C01783=1043.976,340.554,-119.354,172.680,41.723,158.046
C01784=1043.968,340.306,-119.318,172.674,41.720,158.045
C01785=1043.961,340.060,-119.281,172.670,41.717,158.044
C01786=1043.954,339.812,-119.244,172.665,41.714,158.043
C01787=1043.946,339.565,-119.208,172.660,41.710,158.041
C01788=1043.939,339.317,-119.172,172.656,41.707,158.040
C01789=1043.932,339.070,-119.136,172.650,41.703,158.039
C01790=1043.925,338.823,-119.099,172.646,41.700,158.038
C01791=1043.917,338.576,-119.063,172.641,41.697,158.037
C01792=1043.911,338.328,-119.027,172.636,41.693,158.036
C01793=1043.903,338.081,-118.990,172.631,41.690,158.035
C01794=1043.896,337.834,-118.955,172.627,41.686,158.034
C01795=1043.888,337.587,-118.918,172.622,41.683,158.033
C01796=1043.882,337.340,-118.882,172.618,41.680,158.032
C01797=1043.874,337.092,-118.846,172.612,41.677,158.031
C01798=1043.866,336.845,-118.810,172.608,41.673,158.030
C01799=1043.860,336.598,-118.773,172.603,41.670,158.029
C01800=1043.853,336.350,-118.738,172.599,41.667,158.028
C01801=1043.846,336.103,-118.702,172.593,41.663,158.026
C01802=1043.838,335.855,-118.665,172.589,41.660,158.026
C01803=1043.832,335.608,-118.629,172.584,41.657,158.025
C01804=1043.824,335.361,-118.593,172.580,41.653,158.023
C01805=1043.817,335.114,-118.558,172.575,41.650,158.022
C01806=1043.810,334.866,-118.521,172.571,41.647,158.021
C01807=1043.802,334.619,-118.486,172.565,41.644,158.020
C01808=1043.795,334.371,-118.450,172.561,41.640,158.019
C01809=1043.785,334.043,-118.402,172.555,41.636,158.018
C01810=1043.776,333.714,-118.355,172.549,41.632,158.017
C01811=1043.766,333.386,-118.307,172.543,41.628,158.015
C01812=1043.756,333.058,-118.260,172.537,41.623,158.014
C01813=1043.749,332.811,-118.225,172.532,41.620,158.013
C01814=1043.742,332.564,-118.189,172.528,41.617,158.012
C01815=1043.736,332.315,-118.153,172.522,41.614,158.011
C01816=1043.728,332.069,-118.117,172.518,41.611,158.010
C01817=1043.721,331.821,-118.081,172.514,41.608,158.009
C01818=1043.714,331.573,-118.046,172.509,41.605,158.008
C01819=1043.707,331.326,-118.010,172.505,41.602,158.007
C01820=1043.700,331.078,-117.975,172.500,41.599,158.006
C01821=1043.693,330.832,-117.939,172.495,41.595,158.005
C01822=1043.686,330.584,-117.904,172.491,41.592,158.004
C01823=1043.679,330.336,-117.868,172.486,41.589,158.003
C01824=1043.672,330.090,-117.833,172.482,41.586,158.002
C01825=1043.665,329.842,-117.797,172.478,41.583,158.001
C01826=1043.657,329.594,-117.762,172.473,41.580,158.000
C01827=1043.650,329.347,-117.726,172.469,41.577,157.999
C01828=1043.643,329.100,-117.692,172.465,41.573,157.998
C01829=1043.635,328.852,-117.656,172.459,41.570,157.997
C01830=1043.629,328.605,-117.621,172.456,41.568,157.996
C01831=1043.621,328.358,-117.586,172.450,41.565,157.995
C01832=1043.614,328.110,-117.551,172.446,41.562,157.994
C01833=1043.607,327.862,-117.516,172.442,41.558,157.993
C01834=1043.600,327.615,-117.481,172.437,41.556,157.993
C01835=1043.592,327.367,-117.446,172.433,41.553,157.992
C01836=1043.585,327.120,-117.411,172.429,41.550,157.991
C01837=1043.578,326.873,-117.376,172.424,41.547,157.990
C01838=1043.571,326.625,-117.341,172.420,41.544,157.989
C01839=1043.563,326.378,-117.306,172.416,41.541,157.988
C01840=1043.556,326.130,-117.271,172.411,41.538,157.987
C01841=1043.549,325.883,-117.236,172.407,41.535,157.986
C01842=1043.541,325.635,-117.201,172.403,41.532,157.985
C01843=1043.534,325.388,-117.166,172.398,41.529,157.984
C01844=1043.527,325.141,-117.131,172.393,41.526,157.983
C01845=1043.520,324.893,-117.096,172.389,41.524,157.982
C01846=1043.513,324.646,-117.061,172.384,41.521,157.981
C01847=1043.506,324.398,-117.027,172.380,41.517,157.980
C01848=1043.498,324.151,-116.992,172.376,41.515,157.980
C01849=1043.492,323.903,-116.957,172.372,41.512,157.979
C01850=1043.485,323.656,-116.922,172.367,41.509,157.978
C01851=1043.477,323.409,-116.887,172.363,41.506,157.977
C01852=1043.471,323.161,-116.853,172.359,41.503,157.976
C01853=1043.463,322.914,-116.818,172.355,41.500,157.975
C01854=1043.456,322.666,-116.783,172.350,41.497,157.974
C01855=1043.449,322.418,-116.749,172.346,41.494,157.973
C01856=1043.442,322.171,-116.714,172.342,41.492,157.972
C01857=1043.434,321.924,-116.679,172.338,41.488,157.971
C01858=1043.428,321.676,-116.645,172.333,41.486,157.970
C01859=1043.420,321.429,-116.610,172.329,41.483,157.969
C01860=1043.414,321.181,-116.575,172.325,41.480,157.969
C01861=1043.407,320.933,-116.541,172.321,41.477,157.968
C01862=1043.400,320.686,-116.506,172.317,41.474,157.967
C01863=1043.393,320.438,-116.472,172.312,41.471,157.966
C01864=1043.386,320.191,-116.437,172.308,41.469,157.965
C01865=1043.376,319.858,-116.391,172.302,41.465,157.964
C01866=1043.367,319.524,-116.344,172.297,41.461,157.963
C01867=1043.358,319.191,-116.298,172.291,41.457,157.962
C01868=1043.348,318.858,-116.251,172.285,41.453,157.960
C01869=1043.342,318.611,-116.218,172.281,41.451,157.959
C01870=1043.335,318.363,-116.183,172.277,41.447,157.958
C01871=1043.328,318.116,-116.149,172.273,41.445,157.958
C01872=1043.321,317.868,-116.114,172.268,41.442,157.957
C01873=1043.314,317.621,-116.080,172.264,41.439,157.956
C01874=1043.307,317.373,-116.045,172.260,41.437,157.955
C01875=1043.300,317.126,-116.011,172.256,41.433,157.954
C01876=1043.293,316.878,-115.976,172.252,41.431,157.953
C01877=1043.286,316.630,-115.943,172.248,41.428,157.952
C01878=1043.280,316.383,-115.909,172.244,41.425,157.952
C01879=1043.273,316.136,-115.874,172.240,41.423,157.951
C01880=1043.266,315.888,-115.840,172.236,41.419,157.950
C01881=1043.259,315.640,-115.806,172.231,41.417,157.949
C01882=1043.252,315.392,-115.771,172.227,41.414,157.948
C01883=1043.245,315.145,-115.737,172.223,41.411,157.947
C01884=1043.239,314.898,-115.703,172.219,41.409,157.946
C01885=1043.232,314.650,-115.669,172.215,41.406,157.946
C01886=1043.225,314.402,-115.634,172.211,41.403,157.945
C01887=1043.218,314.154,-115.601,172.207,41.400,157.944
C01888=1043.212,313.908,-115.566,172.204,41.398,157.943
C01889=1043.205,313.660,-115.532,172.200,41.395,157.942
C01890=1043.198,313.412,-115.498,172.196,41.392,157.941
C01891=1043.191,313.164,-115.464,172.192,41.389,157.940
C01892=1043.185,312.917,-115.430,172.188,41.387,157.940
C01893=1043.178,312.669,-115.396,172.184,41.383,157.939
C01894=1043.171,312.422,-115.362,172.180,41.381,157.938
C01895=1043.164,312.175,-115.329,172.176,41.378,157.937
C01896=1043.157,311.927,-115.295,172.171,41.376,157.936
C01897=1043.150,311.679,-115.261,172.167,41.373,157.935
C01898=1043.143,311.432,-115.227,172.163,41.371,157.935
C01899=1043.136,311.183,-115.194,172.159,41.368,157.934
C01900=1043.129,310.936,-115.161,172.155,41.365,157.933
C01901=1043.122,310.689,-115.127,172.151,41.363,157.932
C01902=1043.115,310.441,-115.093,172.147,41.360,157.931
C01903=1043.108,310.193,-115.060,172.143,41.358,157.931
C01904=1043.101,309.946,-115.027,172.140,41.355,157.930
C01905=1043.093,309.698,-114.993,172.136,41.352,157.929
C01906=1043.086,309.451,-114.959,172.132,41.350,157.928
C01907=1043.080,309.203,-114.927,172.128,41.348,157.927
C01908=1043.073,308.955,-114.893,172.124,41.345,157.927
C01909=1043.066,308.708,-114.859,172.120,41.343,157.926
C01910=1043.059,308.459,-114.826,172.116,41.340,157.925
C01911=1043.052,308.212,-114.792,172.112,41.337,157.924
C01912=1043.044,307.965,-114.759,172.108,41.335,157.923
C01913=1043.038,307.718,-114.726,172.105,41.332,157.923
C01914=1043.031,307.470,-114.693,172.101,41.330,157.922
C01915=1043.024,307.222,-114.659,172.097,41.327,157.921
C01916=1043.017,306.975,-114.626,172.093,41.325,157.920
C01917=1043.010,306.726,-114.593,172.089,41.322,157.920
C01918=1043.003,306.479,-114.559,172.085,41.320,157.919
C01919=1042.996,306.232,-114.526,172.081,41.317,157.918
C01920=1042.989,305.984,-114.493,172.077,41.314,157.917
C01921=1042.980,305.655,-114.449,172.072,41.311,157.916
C01922=1042.971,305.326,-114.405,172.067,41.308,157.915
C01923=1042.962,304.998,-114.361,172.062,41.305,157.914
C01924=1042.953,304.669,-114.317,172.057,41.302,157.913
C01925=1042.946,304.422,-114.284,172.053,41.299,157.912
C01926=1042.939,304.174,-114.251,172.049,41.296,157.911
C01927=1042.933,303.926,-114.218,172.045,41.294,157.911
C01928=1042.925,303.679,-114.185,172.041,41.291,157.910
C01929=1042.919,303.431,-114.152,172.038,41.289,157.909
C01930=1042.912,303.183,-114.119,172.034,41.286,157.908
C01931=1042.905,302.936,-114.085,172.030,41.284,157.908
C01932=1042.898,302.688,-114.052,172.026,41.281,157.907
C01933=1042.892,302.440,-114.019,172.023,41.279,157.906
C01934=1042.884,302.193,-113.986,172.019,41.277,157.905
C01935=1042.878,301.945,-113.954,172.015,41.274,157.905
C01936=1042.871,301.697,-113.921,172.011,41.271,157.904
C01937=1042.864,301.449,-113.888,172.008,41.269,157.903
C01938=1042.858,301.202,-113.854,172.004,41.267,157.902
C01939=1042.850,300.954,-113.822,172.000,41.264,157.902
C01940=1042.844,300.707,-113.789,171.996,41.261,157.901
C01941=1042.838,300.459,-113.756,171.992,41.259,157.900
C01942=1042.831,300.211,-113.723,171.989,41.257,157.899
C01943=1042.824,299.963,-113.690,171.985,41.254,157.899
C01944=1042.816,299.716,-113.657,171.982,41.252,157.898
C01945=1042.810,299.468,-113.624,171.978,41.249,157.897
C01946=1042.804,299.221,-113.592,171.974,41.247,157.896
C01947=1042.797,298.972,-113.559,171.970,41.244,157.895
C01948=1042.791,298.725,-113.526,171.967,41.242,157.895
C01949=1042.784,298.477,-113.494,171.963,41.239,157.894
C01950=1042.777,298.229,-113.461,171.960,41.237,157.893
C01951=1042.770,297.981,-113.428,171.956,41.235,157.893
C01952=1042.764,297.734,-113.395,171.952,41.232,157.892
C01953=1042.758,297.486,-113.362,171.948,41.229,157.891
C01954=1042.750,297.238,-113.330,171.945,41.227,157.890
C01955=1042.744,296.991,-113.297,171.941,41.225,157.890
C01956=1042.738,296.743,-113.264,171.938,41.223,157.889
C01957=1042.731,296.496,-113.232,171.934,41.220,157.888
C01958=1042.724,296.248,-113.199,171.930,41.217,157.887
C01959=1042.717,296.000,-113.166,171.927,41.215,157.887
C01960=1042.711,295.752,-113.134,171.923,41.213,157.886
C01961=1042.705,295.504,-113.102,171.919,41.210,157.885
C01962=1042.698,295.256,-113.069,171.916,41.208,157.884
C01963=1042.691,295.009,-113.037,171.913,41.206,157.884
C01964=1042.684,294.761,-113.004,171.909,41.203,157.883
C01965=1042.678,294.513,-112.973,171.905,41.201,157.882
C01966=1042.671,294.265,-112.940,171.901,41.198,157.882
C01967=1042.664,294.018,-112.907,171.898,41.196,157.881
C01968=1042.658,293.770,-112.875,171.895,41.194,157.880
C01969=1042.651,293.522,-112.843,171.891,41.192,157.879
C01970=1042.644,293.274,-112.810,171.887,41.189,157.879
C01971=1042.637,293.026,-112.779,171.884,41.187,157.878
C01972=1042.630,292.779,-112.747,171.881,41.185,157.877
C01973=1042.624,292.531,-112.714,171.877,41.182,157.877
C01974=1042.616,292.283,-112.682,171.873,41.180,157.876
C01975=1042.609,292.035,-112.650,171.869,41.177,157.875
C01976=1042.603,291.787,-112.618,171.866,41.175,157.875
C01977=1042.594,291.475,-112.577,171.862,41.173,157.874
C01978=1042.586,291.163,-112.538,171.858,41.170,157.873
C01979=1042.578,290.851,-112.497,171.853,41.167,157.872
C01980=1042.569,290.539,-112.456,171.849,41.164,157.871
C01981=1042.562,290.290,-112.424,171.845,41.162,157.870
C01982=1042.556,290.042,-112.392,171.841,41.159,157.870
C01983=1042.549,289.795,-112.360,171.837,41.157,157.869
C01984=1042.542,289.547,-112.329,171.835,41.155,157.868
C01985=1042.535,289.300,-112.297,171.831,41.153,157.868
C01986=1042.529,289.052,-112.265,171.827,41.150,157.867
C01987=1042.522,288.804,-112.233,171.824,41.148,157.866
C01988=1042.515,288.556,-112.201,171.821,41.146,157.866
C01989=1042.508,288.308,-112.169,171.817,41.143,157.865
C01990=1042.501,288.060,-112.138,171.814,41.141,157.864
C01991=1042.495,287.812,-112.105,171.810,41.139,157.864
C01992=1042.488,287.564,-112.074,171.807,41.137,157.863
C01993=1042.482,287.316,-112.042,171.803,41.135,157.862
C01994=1042.475,287.069,-112.011,171.800,41.132,157.861
C01995=1042.468,286.821,-111.979,171.796,41.130,157.861
C01996=1042.461,286.573,-111.947,171.793,41.128,157.860
C01997=1042.454,286.325,-111.916,171.790,41.126,157.860
C01998=1042.448,286.077,-111.884,171.786,41.123,157.859
C01999=1042.442,285.829,-111.852,171.782,41.121,157.858
C02000=1042.434,285.581,-111.821,171.780,41.119,157.857
C02001=1042.427,285.333,-111.788,171.776,41.117,157.857
C02002=1042.421,285.086,-111.757,171.772,41.115,157.856
C02003=1042.414,284.838,-111.725,171.770,41.113,157.856
C02004=1042.407,284.590,-111.694,171.766,41.110,157.855
C02005=1042.400,284.342,-111.663,171.762,41.108,157.854
C02006=1042.394,284.094,-111.631,171.759,41.106,157.854
C02007=1042.387,283.846,-111.600,171.755,41.104,157.853
C02008=1042.380,283.598,-111.568,171.752,41.102,157.852
C02009=1042.373,283.350,-111.537,171.749,41.100,157.852
C02010=1042.367,283.102,-111.505,171.745,41.098,157.851
C02011=1042.360,282.854,-111.474,171.743,41.096,157.850
C02012=1042.353,282.607,-111.443,171.739,41.093,157.850
C02013=1042.347,282.359,-111.411,171.735,41.091,157.849
C02014=1042.340,282.111,-111.380,171.732,41.089,157.848
C02015=1042.333,281.863,-111.348,171.729,41.087,157.848
C02016=1042.326,281.615,-111.317,171.726,41.084,157.847
C02017=1042.320,281.366,-111.286,171.722,41.082,157.846
C02018=1042.314,281.119,-111.255,171.719,41.080,157.846
C02019=1042.307,280.871,-111.224,171.716,41.078,157.845
C02020=1042.300,280.623,-111.192,171.712,41.076,157.844
C02021=1042.294,280.376,-111.161,171.709,41.073,157.844
C02022=1042.287,280.128,-111.129,171.706,41.071,157.843
C02023=1042.280,279.880,-111.098,171.702,41.069,157.842
C02024=1042.274,279.631,-111.067,171.699,41.067,157.842
C02025=1042.267,279.383,-111.036,171.695,41.065,157.841
C02026=1042.260,279.135,-111.004,171.693,41.063,157.841
C02027=1042.254,278.888,-110.973,171.689,41.061,157.840
C02028=1042.248,278.640,-110.943,171.686,41.059,157.839
C02029=1042.240,278.392,-110.912,171.683,41.057,157.839
C02030=1042.234,278.144,-110.880,171.679,41.054,157.838
C02031=1042.227,277.896,-110.850,171.676,41.052,157.837
C02032=1042.220,277.648,-110.818,171.673,41.050,157.837
C02033=1042.212,277.348,-110.781,171.669,41.048,157.836
C02034=1042.204,277.047,-110.743,171.665,41.045,157.835
C02035=1042.196,276.747,-110.706,171.661,41.043,157.834
C02036=1042.187,276.446,-110.669,171.657,41.040,157.834
C02037=1042.181,276.198,-110.637,171.654,41.038,157.833
C02038=1042.175,275.950,-110.607,171.651,41.036,157.832
C02039=1042.168,275.702,-110.575,171.647,41.034,157.832
C02040=1042.161,275.454,-110.545,171.644,41.032,157.831
C02041=1042.154,275.206,-110.514,171.641,41.030,157.831
C02042=1042.148,274.958,-110.483,171.638,41.027,157.830
C02043=1042.142,274.710,-110.452,171.634,41.025,157.829
C02044=1042.135,274.462,-110.422,171.632,41.023,157.829
C02045=1042.128,274.214,-110.391,171.628,41.021,157.828
C02046=1042.121,273.966,-110.360,171.625,41.020,157.828
C02047=1042.114,273.718,-110.329,171.622,41.017,157.827
C02048=1042.108,273.470,-110.299,171.619,41.015,157.826
C02049=1042.101,273.223,-110.268,171.615,41.013,157.826
C02050=1042.094,272.974,-110.237,171.613,41.011,157.825
C02051=1042.088,272.726,-110.206,171.609,41.009,157.824
C02052=1042.081,272.479,-110.176,171.606,41.007,157.824
C02053=1042.075,272.230,-110.145,171.603,41.005,157.823
C02054=1042.068,271.982,-110.114,171.600,41.003,157.822
C02055=1042.061,271.734,-110.084,171.596,41.001,157.822
C02056=1042.055,271.486,-110.053,171.594,40.999,157.821
C02057=1042.049,271.238,-110.023,171.591,40.997,157.821
C02058=1042.041,270.990,-109.992,171.587,40.995,157.820
C02059=1042.035,270.742,-109.961,171.585,40.992,157.819
C02060=1042.028,270.494,-109.931,171.581,40.990,157.819
C02061=1042.022,270.246,-109.901,171.578,40.989,157.818
C02062=1042.014,269.998,-109.870,171.575,40.987,157.818
C02063=1042.009,269.750,-109.840,171.572,40.984,157.817
C02064=1042.001,269.502,-109.809,171.568,40.982,157.816
C02065=1041.995,269.254,-109.778,171.566,40.980,157.816
C02066=1041.988,269.005,-109.748,171.562,40.979,157.815
C02067=1041.982,268.758,-109.718,171.559,40.977,157.815
C02068=1041.975,268.509,-109.688,171.557,40.974,157.814
C02069=1041.968,268.261,-109.658,171.553,40.972,157.813
C02070=1041.962,268.013,-109.627,171.550,40.970,157.813
C02071=1041.955,267.765,-109.597,171.547,40.969,157.812
C02072=1041.949,267.517,-109.567,171.544,40.966,157.812
C02073=1041.942,267.269,-109.537,171.540,40.964,157.811
C02074=1041.935,267.021,-109.506,171.538,40.962,157.811
C02075=1041.929,266.773,-109.476,171.535,40.961,157.810
C02076=1041.921,266.525,-109.446,171.531,40.959,157.809
C02077=1041.915,266.276,-109.415,171.529,40.956,157.809
C02078=1041.908,266.029,-109.386,171.525,40.954,157.808
C02079=1041.901,265.781,-109.356,171.523,40.953,157.808
C02080=1041.895,265.532,-109.325,171.520,40.950,157.807
C02081=1041.888,265.285,-109.295,171.516,40.948,157.806
C02082=1041.881,265.036,-109.265,171.514,40.946,157.806
C02083=1041.875,264.788,-109.235,171.510,40.945,157.805
C02084=1041.868,264.540,-109.205,171.507,40.943,157.805
C02085=1041.861,264.292,-109.174,171.505,40.940,157.804
C02086=1041.855,264.044,-109.144,171.501,40.939,157.804
C02087=1041.848,263.795,-109.115,171.498,40.937,157.803
C02088=1041.842,263.548,-109.085,171.496,40.934,157.802
C02089=1041.833,263.252,-109.048,171.492,40.932,157.802
C02090=1041.826,262.956,-109.013,171.488,40.930,157.801
C02091=1041.818,262.660,-108.977,171.484,40.928,157.800
C02092=1041.810,262.364,-108.941,171.481,40.925,157.800
C02093=1041.803,262.116,-108.912,171.478,40.923,157.799
C02094=1041.797,261.868,-108.882,171.475,40.921,157.798
C02095=1041.790,261.620,-108.852,171.472,40.920,157.798
C02096=1041.783,261.372,-108.823,171.469,40.917,157.797
C02097=1041.776,261.123,-108.793,171.466,40.916,157.797
C02098=1041.769,260.875,-108.763,171.463,40.914,157.796
C02099=1041.763,260.627,-108.733,171.461,40.912,157.796
C02100=1041.756,260.379,-108.703,171.457,40.910,157.795
C02101=1041.750,260.131,-108.674,171.454,40.908,157.794
C02102=1041.742,259.883,-108.644,171.452,40.906,157.794
C02103=1041.736,259.634,-108.615,171.448,40.904,157.793
C02104=1041.729,259.386,-108.585,171.445,40.903,157.793
C02105=1041.723,259.138,-108.556,171.443,40.900,157.792
C02106=1041.715,258.890,-108.526,171.439,40.899,157.792
C02107=1041.708,258.641,-108.497,171.437,40.897,157.791
C02108=1041.701,258.394,-108.467,171.434,40.895,157.791
C02109=1041.695,258.145,-108.438,171.430,40.893,157.790
C02110=1041.688,257.898,-108.408,171.428,40.891,157.790
C02111=1041.681,257.649,-108.379,171.425,40.889,157.789
C02112=1041.675,257.401,-108.349,171.422,40.888,157.788
C02113=1041.668,257.153,-108.320,171.419,40.886,157.788
C02114=1041.661,256.905,-108.290,171.416,40.884,157.787
C02115=1041.655,256.657,-108.261,171.413,40.882,157.787
C02116=1041.648,256.408,-108.231,171.410,40.880,157.786
C02117=1041.642,256.160,-108.202,171.408,40.878,157.786
C02118=1041.635,255.912,-108.172,171.405,40.876,157.785
C02119=1041.627,255.664,-108.143,171.401,40.874,157.785
C02120=1041.621,255.415,-108.114,171.399,40.872,157.784
C02121=1041.614,255.167,-108.085,171.396,40.871,157.784
C02122=1041.608,254.920,-108.055,171.393,40.868,157.783
C02123=1041.601,254.671,-108.025,171.390,40.867,157.782
C02124=1041.595,254.423,-107.996,171.387,40.865,157.782
C02125=1041.587,254.175,-107.966,171.385,40.863,157.781
C02126=1041.581,253.927,-107.937,171.382,40.861,157.781
C02127=1041.575,253.678,-107.908,171.379,40.859,157.780
C02128=1041.568,253.430,-107.879,171.376,40.857,157.780
C02129=1041.562,253.182,-107.849,171.373,40.855,157.779
C02130=1041.554,252.934,-107.820,171.371,40.853,157.779
C02131=1041.548,252.685,-107.791,171.367,40.852,157.778
C02132=1041.541,252.437,-107.762,171.365,40.850,157.777
C02133=1041.535,252.188,-107.733,171.362,40.847,157.777
C02134=1041.528,251.941,-107.703,171.359,40.846,157.776
C02135=1041.522,251.693,-107.674,171.356,40.844,157.776
C02136=1041.515,251.444,-107.644,171.353,40.842,157.775
C02137=1041.509,251.196,-107.615,171.350,40.840,157.775
C02138=1041.502,250.948,-107.587,171.348,40.838,157.774
C02139=1041.495,250.701,-107.557,171.345,40.836,157.774
C02140=1041.488,250.452,-107.528,171.342,40.835,157.773
C02141=1041.482,250.204,-107.499,171.339,40.832,157.772
C02142=1041.476,249.955,-107.470,171.337,40.831,157.772
C02143=1041.469,249.707,-107.440,171.334,40.828,157.771
C02144=1041.463,249.458,-107.411,171.331,40.827,157.771
C02145=1041.455,249.161,-107.376,171.328,40.824,157.770
C02146=1041.447,248.864,-107.342,171.324,40.822,157.770
C02147=1041.439,248.567,-107.307,171.321,40.820,157.769
C02148=1041.431,248.269,-107.272,171.318,40.818,157.768
C02149=1041.425,248.021,-107.243,171.315,40.816,157.768
C02150=1041.418,247.772,-107.214,171.312,40.814,157.767
C02151=1041.412,247.524,-107.185,171.310,40.812,157.767
C02152=1041.406,247.276,-107.156,171.307,40.810,157.766
C02153=1041.399,247.028,-107.127,171.304,40.808,157.766
C02154=1041.392,246.780,-107.098,171.301,40.806,157.765
C02155=1041.386,246.531,-107.069,171.298,40.804,157.764
C02156=1041.380,246.283,-107.040,171.296,40.802,157.764
C02157=1041.373,246.035,-107.011,171.293,40.800,157.763
C02158=1041.367,245.787,-106.982,171.290,40.798,157.763
C02159=1041.360,245.539,-106.953,171.288,40.796,157.762
C02160=1041.353,245.290,-106.924,171.285,40.794,157.762
C02161=1041.347,245.042,-106.896,171.283,40.793,157.761
C02162=1041.341,244.793,-106.866,171.279,40.791,157.761
C02163=1041.334,244.546,-106.838,171.277,40.789,157.760
C02164=1041.328,244.298,-106.809,171.274,40.787,157.759
C02165=1041.320,244.049,-106.780,171.271,40.785,157.759
C02166=1041.314,243.800,-106.752,171.269,40.783,157.759
C02167=1041.308,243.552,-106.723,171.266,40.781,157.758
C02168=1041.301,243.304,-106.694,171.264,40.780,157.757
C02169=1041.295,243.056,-106.665,171.261,40.777,157.757
C02170=1041.288,242.808,-106.638,171.259,40.776,157.756
C02171=1041.281,242.559,-106.608,171.255,40.774,157.756
C02172=1041.275,242.311,-106.579,171.252,40.772,157.755
C02173=1041.268,242.062,-106.551,171.250,40.770,157.755
C02174=1041.262,241.814,-106.522,171.247,40.768,157.754
C02175=1041.255,241.566,-106.494,171.245,40.767,157.754
C02176=1041.249,241.318,-106.466,171.242,40.764,157.753
C02177=1041.242,241.070,-106.437,171.240,40.763,157.753
C02178=1041.235,240.821,-106.408,171.237,40.761,157.752
C02179=1041.229,240.573,-106.380,171.234,40.759,157.752
C02180=1041.222,240.324,-106.351,171.232,40.757,157.751
C02181=1041.216,240.076,-106.323,171.229,40.755,157.751
C02182=1041.209,239.828,-106.295,171.226,40.754,157.750
C02183=1041.203,239.579,-106.266,171.223,40.752,157.750
C02184=1041.196,239.332,-106.238,171.221,40.750,157.749
C02185=1041.188,239.082,-106.210,171.218,40.748,157.749
C02186=1041.182,238.834,-106.181,171.215,40.747,157.748
C02187=1041.176,238.586,-106.153,171.213,40.744,157.747
C02188=1041.169,238.338,-106.125,171.210,40.743,157.747
C02189=1041.163,238.089,-106.096,171.208,40.741,157.747
C02190=1041.156,237.841,-106.068,171.205,40.739,157.746
C02191=1041.149,237.593,-106.040,171.203,40.737,157.745
C02192=1041.143,237.345,-106.011,171.200,40.736,157.745
C02193=1041.136,237.096,-105.983,171.197,40.733,157.744
C02194=1041.129,236.848,-105.956,171.195,40.732,157.744
C02195=1041.122,236.600,-105.927,171.192,40.730,157.743
C02196=1041.116,236.351,-105.899,171.190,40.728,157.743
C02197=1041.109,236.103,-105.870,171.187,40.726,157.742
C02198=1041.102,235.854,-105.842,171.185,40.725,157.742
C02199=1041.095,235.606,-105.815,171.181,40.723,157.741
C02200=1041.089,235.358,-105.786,171.179,40.721,157.741
C02201=1041.081,235.054,-105.752,171.176,40.719,157.740
C02202=1041.073,234.752,-105.718,171.173,40.716,157.740
C02203=1041.065,234.449,-105.684,171.170,40.714,157.739
C02204=1041.057,234.146,-105.649,171.167,40.712,157.738
C02205=1041.051,233.897,-105.621,171.164,40.710,157.738
C02206=1041.044,233.649,-105.593,171.162,40.708,157.737
C02207=1041.037,233.401,-105.565,171.159,40.707,157.737
C02208=1041.031,233.152,-105.537,171.157,40.704,157.736
C02209=1041.025,232.904,-105.509,171.154,40.703,157.736
C02210=1041.018,232.655,-105.481,171.152,40.701,157.735
C02211=1041.011,232.407,-105.452,171.149,40.699,157.735
C02212=1041.004,232.159,-105.425,171.147,40.697,157.734
C02213=1040.998,231.910,-105.396,171.144,40.696,157.734
C02214=1040.992,231.662,-105.369,171.141,40.693,157.733
C02215=1040.985,231.413,-105.341,171.139,40.692,157.733
C02216=1040.978,231.165,-105.313,171.136,40.690,157.732
C02217=1040.972,230.916,-105.286,171.134,40.688,157.732
C02218=1040.965,230.669,-105.257,171.131,40.686,157.731
C02219=1040.958,230.420,-105.229,171.129,40.685,157.731
C02220=1040.951,230.172,-105.202,171.126,40.682,157.730
C02221=1040.945,229.923,-105.174,171.124,40.681,157.730
C02222=1040.939,229.675,-105.146,171.121,40.679,157.729
C02223=1040.932,229.426,-105.118,171.118,40.677,157.729
C02224=1040.925,229.178,-105.090,171.116,40.675,157.728
C02225=1040.919,228.929,-105.062,171.113,40.674,157.728
C02226=1040.913,228.681,-105.035,171.111,40.672,157.727
C02227=1040.906,228.433,-105.007,171.108,40.670,157.727
C02228=1040.899,228.185,-104.980,171.106,40.668,157.726
C02229=1040.893,227.936,-104.952,171.103,40.667,157.726
C02230=1040.886,227.688,-104.924,171.102,40.665,157.725
C02231=1040.879,227.439,-104.896,171.099,40.663,157.725
C02232=1040.872,227.191,-104.869,171.097,40.661,157.724
C02233=1040.865,226.943,-104.841,171.094,40.659,157.724
C02234=1040.858,226.694,-104.814,171.092,40.658,157.723
C02235=1040.852,226.445,-104.787,171.089,40.655,157.723
C02236=1040.845,226.197,-104.759,171.086,40.654,157.722
C02237=1040.839,225.948,-104.731,171.084,40.652,157.722
C02238=1040.833,225.701,-104.704,171.081,40.651,157.721
C02239=1040.826,225.452,-104.676,171.079,40.648,157.721
C02240=1040.818,225.204,-104.649,171.076,40.647,157.720
C02241=1040.812,224.956,-104.621,171.074,40.645,157.720
C02242=1040.805,224.706,-104.594,171.071,40.643,157.719
C02243=1040.799,224.458,-104.567,171.070,40.641,157.719
C02244=1040.792,224.210,-104.539,171.067,40.639,157.718
C02245=1040.785,223.961,-104.511,171.065,40.638,157.718
C02246=1040.779,223.713,-104.484,171.062,40.636,157.717
C02247=1040.772,223.465,-104.457,171.060,40.634,157.717
C02248=1040.766,223.216,-104.430,171.057,40.632,157.716
C02249=1040.759,222.968,-104.402,171.055,40.631,157.716
C02250=1040.752,222.719,-104.374,171.052,40.629,157.715
C02251=1040.746,222.471,-104.347,171.049,40.627,157.715
C02252=1040.740,222.223,-104.320,171.048,40.625,157.714
C02253=1040.732,221.974,-104.293,171.045,40.623,157.714
C02254=1040.726,221.725,-104.266,171.043,40.621,157.713
C02255=1040.719,221.477,-104.238,171.040,40.620,157.713
C02256=1040.713,221.229,-104.211,171.038,40.618,157.712
C02257=1040.704,220.918,-104.176,171.035,40.616,157.712
C02258=1040.697,220.608,-104.142,171.032,40.613,157.711
C02259=1040.688,220.297,-104.108,171.029,40.611,157.711
C02260=1040.680,219.987,-104.074,171.026,40.608,157.710
C02261=1040.674,219.738,-104.047,171.024,40.607,157.709
C02262=1040.666,219.490,-104.020,171.021,40.605,157.709
C02263=1040.660,219.240,-103.993,171.019,40.603,157.708
C02264=1040.653,218.992,-103.965,171.017,40.602,157.708
C02265=1040.647,218.745,-103.939,171.015,40.600,157.708
C02266=1040.640,218.496,-103.912,171.012,40.598,157.707
C02267=1040.633,218.247,-103.884,171.009,40.596,157.706
C02268=1040.626,217.998,-103.857,171.007,40.595,157.706
C02269=1040.620,217.751,-103.831,171.004,40.593,157.706
C02270=1040.613,217.502,-103.804,171.003,40.591,157.705
C02271=1040.607,217.253,-103.777,171.000,40.589,157.705
C02272=1040.599,217.005,-103.749,170.998,40.587,157.704
C02273=1040.594,216.756,-103.723,170.995,40.586,157.704
C02274=1040.586,216.508,-103.696,170.993,40.584,157.703
C02275=1040.580,216.259,-103.669,170.991,40.582,157.703
C02276=1040.572,216.011,-103.642,170.989,40.580,157.702
C02277=1040.567,215.763,-103.615,170.986,40.578,157.702
C02278=1040.560,215.514,-103.588,170.984,40.577,157.701
C02279=1040.553,215.265,-103.561,170.981,40.575,157.701
C02280=1040.547,215.017,-103.534,170.980,40.573,157.700
C02281=1040.540,214.769,-103.507,170.977,40.571,157.700
C02282=1040.533,214.520,-103.480,170.975,40.569,157.699
C02283=1040.527,214.272,-103.454,170.972,40.568,157.699
C02284=1040.520,214.023,-103.426,170.969,40.566,157.698
C02285=1040.513,213.775,-103.400,170.968,40.564,157.698
C02286=1040.507,213.526,-103.373,170.965,40.562,157.697
C02287=1040.500,213.278,-103.345,170.963,40.561,157.697
C02288=1040.493,213.029,-103.319,170.960,40.558,157.696
C02289=1040.488,212.781,-103.292,170.959,40.557,157.696
C02290=1040.480,212.533,-103.265,170.956,40.555,157.695
C02291=1040.474,212.284,-103.238,170.954,40.553,157.695
C02292=1040.467,212.035,-103.212,170.951,40.551,157.694
C02293=1040.461,211.786,-103.185,170.950,40.549,157.694
C02294=1040.454,211.539,-103.158,170.947,40.548,157.693
C02295=1040.448,211.290,-103.131,170.945,40.546,157.693
C02296=1040.441,211.041,-103.105,170.942,40.544,157.692
C02297=1040.434,210.793,-103.079,170.941,40.542,157.692
C02298=1040.428,210.544,-103.052,170.938,40.540,157.691
C02299=1040.420,210.296,-103.025,170.936,40.539,157.691
C02300=1040.415,210.048,-102.998,170.933,40.537,157.691
C02301=1040.407,209.799,-102.972,170.932,40.535,157.690
C02302=1040.401,209.551,-102.946,170.929,40.533,157.689
C02303=1040.395,209.302,-102.919,170.927,40.531,157.689
C02304=1040.387,209.053,-102.892,170.925,40.530,157.689
C02305=1040.381,208.805,-102.866,170.923,40.528,157.688
C02306=1040.375,208.556,-102.839,170.920,40.526,157.688
C02307=1040.368,208.308,-102.813,170.918,40.524,157.687
C02308=1040.361,208.060,-102.786,170.916,40.522,157.687
C02309=1040.353,207.811,-102.759,170.914,40.521,157.686
C02310=1040.348,207.563,-102.733,170.911,40.519,157.686
C02311=1040.341,207.314,-102.706,170.909,40.517,157.685
C02312=1040.334,207.066,-102.680,170.907,40.515,157.685
C02313=1040.326,206.760,-102.648,170.904,40.513,157.684
C02314=1040.318,206.455,-102.616,170.902,40.510,157.684
C02315=1040.310,206.150,-102.583,170.899,40.509,157.683
C02316=1040.301,205.845,-102.551,170.896,40.507,157.682
C02317=1040.275,204.794,-102.445,170.609,40.403,157.648
C02318=1040.269,204.545,-102.419,170.606,40.402,157.648
C02319=1040.263,204.296,-102.394,170.602,40.401,157.647
C02320=1040.256,204.048,-102.369,170.599,40.400,157.647
C02321=1040.250,203.799,-102.343,170.597,40.399,157.647
C02322=1040.245,203.551,-102.318,170.593,40.397,157.646
C02323=1040.239,203.302,-102.294,170.590,40.397,157.646
C02324=1040.233,203.053,-102.268,170.587,40.395,157.646
C02325=1040.226,202.805,-102.244,170.584,40.395,157.645
C02326=1040.219,202.556,-102.218,170.581,40.394,157.645
C02327=1040.213,202.307,-102.193,170.578,40.393,157.645
C02328=1040.208,202.059,-102.169,170.575,40.392,157.644
C02329=1040.202,201.810,-102.143,170.572,40.391,157.644
C02330=1040.195,201.561,-102.118,170.569,40.390,157.644
C02331=1040.189,201.313,-102.093,170.566,40.388,157.643
C02332=1040.183,201.063,-102.068,170.563,40.387,157.643
C02333=1040.176,200.815,-102.043,170.560,40.386,157.643
C02334=1040.170,200.566,-102.018,170.557,40.385,157.642
C02335=1040.165,200.318,-101.994,170.554,40.385,157.642
C02336=1040.158,200.069,-101.969,170.551,40.384,157.642
C02337=1040.152,199.820,-101.944,170.548,40.383,157.641
C02338=1040.145,199.572,-101.920,170.545,40.382,157.641
C02339=1040.139,199.323,-101.895,170.542,40.381,157.641
C02340=1040.133,199.074,-101.870,170.539,40.380,157.640
C02341=1040.127,198.826,-101.846,170.536,40.379,157.640
C02342=1040.121,198.577,-101.821,170.533,40.378,157.640
C02343=1040.114,198.329,-101.796,170.530,40.377,157.639
C02344=1040.108,198.079,-101.771,170.527,40.377,157.639
C02345=1040.101,197.831,-101.747,170.525,40.376,157.639
C02346=1040.096,197.582,-101.722,170.521,40.375,157.638
C02347=1040.090,197.333,-101.698,170.518,40.374,157.638
C02348=1040.083,197.085,-101.673,170.516,40.373,157.638
C02349=1040.077,196.835,-101.648,170.512,40.372,157.637
C02350=1040.070,196.587,-101.624,170.510,40.371,157.637
C02351=1040.065,196.338,-101.599,170.507,40.370,157.637
C02352=1040.058,196.090,-101.575,170.503,40.370,157.637
C02353=1040.052,195.841,-101.550,170.501,40.368,157.636
C02354=1040.046,195.593,-101.526,170.498,40.368,157.636
C02355=1040.040,195.344,-101.501,170.494,40.367,157.636
C02356=1040.033,195.095,-101.477,170.492,40.366,157.635
C02357=1040.027,194.846,-101.452,170.489,40.365,157.635
C02358=1040.021,194.598,-101.427,170.487,40.364,157.635
C02359=1040.015,194.349,-101.403,170.483,40.363,157.634
C02360=1040.009,194.100,-101.378,170.480,40.362,157.634
C02361=1040.003,193.852,-101.354,170.478,40.361,157.634
C02362=1039.997,193.602,-101.330,170.474,40.360,157.633
C02363=1039.990,193.354,-101.305,170.472,40.360,157.633
C02364=1039.984,193.105,-101.281,170.469,40.359,157.633
C02365=1039.978,192.856,-101.257,170.466,40.358,157.633
C02366=1039.972,192.607,-101.232,170.463,40.357,157.632
C02367=1039.966,192.360,-101.208,170.460,40.356,157.632
C02368=1039.960,192.110,-101.183,170.458,40.356,157.632
C02369=1039.953,191.861,-101.159,170.454,40.355,157.631
C02370=1039.948,191.613,-101.135,170.452,40.354,157.631
C02371=1039.941,191.364,-101.110,170.449,40.353,157.631
C02372=1039.935,191.116,-101.086,170.445,40.352,157.630
C02373=1039.929,190.867,-101.062,170.443,40.351,157.630
C02374=1039.923,190.617,-101.037,170.440,40.350,157.630
C02375=1039.918,190.369,-101.013,170.438,40.349,157.630
C02376=1039.911,190.121,-100.988,170.434,40.348,157.629
C02377=1039.905,189.872,-100.964,170.432,40.348,157.629
C02378=1039.898,189.587,-100.936,170.429,40.347,157.629
C02379=1039.891,189.303,-100.908,170.425,40.346,157.628
C02380=1039.884,189.018,-100.881,170.422,40.345,157.628
C02381=1039.877,188.734,-100.853,170.419,40.344,157.628
C02382=1039.871,188.485,-100.829,170.416,40.343,157.627
C02383=1039.865,188.237,-100.805,170.413,40.342,157.627
C02384=1039.859,187.988,-100.780,170.411,40.341,157.627
C02385=1039.853,187.739,-100.757,170.408,40.341,157.627
C02386=1039.847,187.490,-100.732,170.405,40.340,157.626
C02387=1039.841,187.242,-100.708,170.402,40.339,157.626
C02388=1039.835,186.992,-100.684,170.400,40.338,157.626
C02389=1039.829,186.744,-100.660,170.396,40.337,157.625
C02390=1039.824,186.495,-100.636,170.394,40.336,157.625
C02391=1039.817,186.247,-100.612,170.391,40.335,157.625
C02392=1039.812,185.997,-100.587,170.388,40.334,157.624
C02393=1039.806,185.749,-100.564,170.385,40.334,157.624
C02394=1039.799,185.500,-100.540,170.383,40.333,157.624
C02395=1039.794,185.252,-100.515,170.380,40.332,157.624
C02396=1039.787,185.003,-100.491,170.377,40.332,157.623
C02397=1039.782,184.754,-100.467,170.374,40.331,157.623
C02398=1039.775,184.505,-100.443,170.372,40.330,157.623
C02399=1039.770,184.256,-100.419,170.369,40.329,157.622
C02400=1039.764,184.008,-100.395,170.366,40.328,157.622
C02401=1039.758,183.759,-100.371,170.363,40.327,157.622
C02402=1039.752,183.511,-100.347,170.361,40.326,157.622
C02403=1039.745,183.261,-100.324,170.358,40.326,157.621
C02404=1039.739,183.013,-100.300,170.355,40.325,157.621
C02405=1039.733,182.764,-100.276,170.352,40.325,157.621
C02406=1039.727,182.515,-100.252,170.350,40.324,157.621
C02407=1039.720,182.266,-100.229,170.347,40.323,157.620
C02408=1039.714,182.018,-100.205,170.344,40.323,157.620
C02409=1039.708,181.769,-100.181,170.341,40.322,157.620
C02410=1039.702,181.520,-100.158,170.339,40.321,157.620
C02411=1039.695,181.271,-100.135,170.336,40.321,157.619
C02412=1039.689,181.023,-100.111,170.333,40.320,157.619
C02413=1039.682,180.773,-100.088,170.330,40.320,157.619
C02414=1039.676,180.525,-100.064,170.328,40.319,157.619
C02415=1039.670,180.276,-100.040,170.325,40.318,157.618
C02416=1039.664,180.027,-100.017,170.323,40.318,157.618
C02417=1039.657,179.778,-99.993,170.319,40.317,157.618
C02418=1039.651,179.529,-99.970,170.317,40.316,157.618
C02419=1039.645,179.280,-99.946,170.314,40.316,157.618
C02420=1039.639,179.032,-99.923,170.312,40.315,157.617
C02421=1039.632,178.783,-99.900,170.308,40.315,157.617
C02422=1039.626,178.534,-99.876,170.306,40.314,157.617
C02423=1039.620,178.285,-99.853,170.303,40.313,157.617
C02424=1039.613,178.036,-99.829,170.301,40.313,157.616
C02425=1039.608,177.788,-99.806,170.297,40.313,157.616
C02426=1039.601,177.539,-99.782,170.295,40.312,157.616
C02427=1039.595,177.290,-99.759,170.292,40.311,157.616
C02428=1039.589,177.041,-99.736,170.290,40.310,157.615
C02429=1039.583,176.792,-99.712,170.288,40.310,157.615
C02430=1039.576,176.544,-99.689,170.284,40.309,157.615
C02431=1039.570,176.294,-99.666,170.282,40.308,157.615
C02432=1039.564,176.046,-99.642,170.279,40.308,157.614
C02433=1039.558,175.797,-99.619,170.277,40.308,157.614
C02434=1039.551,175.548,-99.595,170.273,40.307,157.614
C02435=1039.546,175.299,-99.572,170.271,40.306,157.614
C02436=1039.540,175.050,-99.549,170.268,40.306,157.614
C02437=1039.533,174.801,-99.525,170.266,40.305,157.613
C02438=1039.527,174.553,-99.503,170.264,40.304,157.613
C02439=1039.521,174.304,-99.479,170.260,40.304,157.613
C02440=1039.514,174.055,-99.456,170.258,40.303,157.613
C02441=1039.509,173.806,-99.433,170.255,40.303,157.612
C02442=1039.502,173.521,-99.406,170.253,40.302,157.612
C02443=1039.495,173.237,-99.380,170.249,40.301,157.612
C02444=1039.488,172.952,-99.353,170.246,40.301,157.612
C02445=1039.481,172.667,-99.327,170.243,40.300,157.611
C02446=1039.474,172.418,-99.303,170.241,40.300,157.611
C02447=1039.468,172.169,-99.280,170.238,40.299,157.611
C02448=1039.463,171.921,-99.257,170.235,40.298,157.611
C02449=1039.456,171.672,-99.235,170.233,40.298,157.610
C02450=1039.450,171.423,-99.211,170.230,40.297,157.610
C02451=1039.444,171.174,-99.188,170.227,40.296,157.610
C02452=1039.438,170.925,-99.165,170.225,40.296,157.610
C02453=1039.432,170.676,-99.142,170.222,40.295,157.609
C02454=1039.426,170.427,-99.118,170.220,40.295,157.609
C02455=1039.420,170.178,-99.095,170.217,40.294,157.609
C02456=1039.414,169.930,-99.073,170.214,40.294,157.609
C02457=1039.408,169.681,-99.050,170.212,40.293,157.608
C02458=1039.401,169.432,-99.026,170.209,40.293,157.608
C02459=1039.395,169.183,-99.003,170.207,40.292,157.608
C02460=1039.390,168.934,-98.980,170.205,40.291,157.608
C02461=1039.383,168.686,-98.957,170.201,40.291,157.608
C02462=1039.378,168.437,-98.934,170.199,40.290,157.607
C02463=1039.371,168.188,-98.911,170.197,40.289,157.607
C02464=1039.365,167.939,-98.887,170.194,40.289,157.607
C02465=1039.359,167.690,-98.864,170.191,40.288,157.607
C02466=1039.354,167.441,-98.842,170.189,40.288,157.607
C02467=1039.347,167.192,-98.819,170.186,40.287,157.606
C02468=1039.342,166.944,-98.796,170.184,40.287,157.606
C02469=1039.336,166.695,-98.773,170.182,40.286,157.606
C02470=1039.329,166.445,-98.750,170.178,40.285,157.605
C02471=1039.324,166.196,-98.727,170.176,40.285,157.605
C02472=1039.317,165.948,-98.704,170.174,40.284,157.605
C02473=1039.311,165.699,-98.681,170.171,40.283,157.605
C02474=1039.305,165.450,-98.658,170.169,40.283,157.605
C02475=1039.300,165.201,-98.635,170.166,40.283,157.604
C02476=1039.294,164.953,-98.612,170.163,40.282,157.604
C02477=1039.288,164.704,-98.590,170.161,40.281,157.604
C02478=1039.282,164.455,-98.567,170.159,40.281,157.604
C02479=1039.275,164.205,-98.544,170.155,40.280,157.604
C02480=1039.270,163.957,-98.521,170.153,40.279,157.603
C02481=1039.264,163.708,-98.498,170.151,40.279,157.603
C02482=1039.258,163.459,-98.475,170.149,40.279,157.603
C02483=1039.252,163.210,-98.452,170.146,40.278,157.603
C02484=1039.246,162.961,-98.429,170.143,40.277,157.602
C02485=1039.240,162.712,-98.406,170.141,40.277,157.602
C02486=1039.234,162.464,-98.384,170.138,40.276,157.602
C02487=1039.228,162.215,-98.361,170.136,40.275,157.602
C02488=1039.222,161.966,-98.338,170.134,40.275,157.601
C02489=1039.217,161.717,-98.315,170.131,40.274,157.601
C02490=1039.211,161.468,-98.293,170.128,40.274,157.601
C02491=1039.205,161.219,-98.271,170.126,40.273,157.601
C02492=1039.199,160.970,-98.248,170.124,40.273,157.601
C02493=1039.193,160.721,-98.225,170.122,40.272,157.600
C02494=1039.188,160.472,-98.202,170.118,40.272,157.600
C02495=1039.181,160.224,-98.180,170.116,40.271,157.600
C02496=1039.175,159.975,-98.157,170.114,40.270,157.600
C02497=1039.169,159.726,-98.135,170.111,40.270,157.600
C02498=1039.164,159.477,-98.112,170.109,40.270,157.599
C02499=1039.157,159.228,-98.090,170.106,40.269,157.599
C02500=1039.151,158.979,-98.067,170.104,40.269,157.599
C02501=1039.145,158.729,-98.045,170.101,40.268,157.599
C02502=1039.138,158.481,-98.022,170.099,40.268,157.599
C02503=1039.132,158.232,-97.999,170.097,40.268,157.598
C02504=1039.126,157.983,-97.978,170.093,40.267,157.598
C02505=1039.120,157.734,-97.955,170.091,40.267,157.598
C02506=1039.113,157.449,-97.930,170.088,40.266,157.598
C02507=1039.106,157.164,-97.904,170.086,40.265,157.598
C02508=1039.100,156.878,-97.879,170.083,40.265,157.597
C02509=1039.092,156.593,-97.853,170.080,40.265,157.597
C02510=1039.086,156.345,-97.830,170.077,40.264,157.597
C02511=1039.080,156.096,-97.809,170.075,40.264,157.597
C02512=1039.074,155.847,-97.786,170.073,40.263,157.597
C02513=1039.068,155.597,-97.764,170.070,40.263,157.596
C02514=1039.062,155.349,-97.741,170.068,40.263,157.596
C02515=1039.056,155.100,-97.719,170.065,40.262,157.596
C02516=1039.049,154.851,-97.697,170.063,40.262,157.596
C02517=1039.044,154.602,-97.674,170.060,40.261,157.596
C02518=1039.038,154.353,-97.653,170.058,40.260,157.595
C02519=1039.031,154.104,-97.630,170.056,40.260,157.595
C02520=1039.025,153.855,-97.609,170.053,40.259,157.595
C02521=1039.019,153.606,-97.586,170.050,40.259,157.595
C02522=1039.013,153.357,-97.564,170.048,40.259,157.595
C02523=1039.007,153.108,-97.542,170.046,40.259,157.595
C02524=1039.000,152.859,-97.520,170.044,40.258,157.594
C02525=1038.994,152.610,-97.498,170.041,40.258,157.594
C02526=1038.989,152.361,-97.476,170.039,40.258,157.594
C02527=1038.982,152.112,-97.453,170.036,40.257,157.594
C02528=1038.976,151.864,-97.432,170.034,40.257,157.594
C02529=1038.970,151.615,-97.410,170.031,40.257,157.593
C02530=1038.964,151.366,-97.388,170.029,40.256,157.593
C02531=1038.958,151.116,-97.366,170.027,40.256,157.593
C02532=1038.952,150.868,-97.343,170.025,40.255,157.593
C02533=1038.946,150.619,-97.322,170.021,40.255,157.593
C02534=1038.939,150.370,-97.299,170.019,40.254,157.593
C02535=1038.933,150.121,-97.278,170.017,40.254,157.592
C02536=1038.928,149.871,-97.256,170.015,40.254,157.592
C02537=1038.921,149.623,-97.233,170.012,40.253,157.592
C02538=1038.915,149.374,-97.212,170.010,40.253,157.592
C02539=1038.910,149.125,-97.190,170.007,40.252,157.592
C02540=1038.903,148.876,-97.168,170.005,40.252,157.591
C02541=1038.897,148.627,-97.146,170.003,40.252,157.591
C02542=1038.891,148.378,-97.125,170.000,40.251,157.591
C02543=1038.885,148.129,-97.102,169.998,40.251,157.591
C02544=1038.879,147.880,-97.080,169.996,40.250,157.591
C02545=1038.873,147.631,-97.058,169.993,40.250,157.591
C02546=1038.867,147.382,-97.037,169.990,40.250,157.590
C02547=1038.861,147.134,-97.015,169.988,40.250,157.590
C02548=1038.854,146.884,-96.993,169.986,40.249,157.590
C02549=1038.848,146.635,-96.972,169.984,40.249,157.590
C02550=1038.842,146.386,-96.950,169.982,40.248,157.590
C02551=1038.836,146.137,-96.928,169.978,40.248,157.590
C02552=1038.830,145.888,-96.906,169.976,40.248,157.589
C02553=1038.823,145.639,-96.884,169.974,40.247,157.589
C02554=1038.818,145.391,-96.863,169.972,40.247,157.589
C02555=1038.812,145.141,-96.841,169.969,40.247,157.589
C02556=1038.805,144.892,-96.820,169.967,40.247,157.589
C02557=1038.799,144.643,-96.799,169.965,40.246,157.589
C02558=1038.792,144.394,-96.777,169.962,40.246,157.588
C02559=1038.786,144.145,-96.755,169.960,40.245,157.588
C02560=1038.780,143.897,-96.733,169.957,40.245,157.588
C02561=1038.774,143.648,-96.712,169.955,40.245,157.588
C02562=1038.768,143.399,-96.690,169.953,40.245,157.588
C02563=1038.762,143.149,-96.669,169.951,40.244,157.588
C02564=1038.756,142.900,-96.647,169.949,40.244,157.587
C02565=1038.750,142.652,-96.626,169.945,40.244,157.587
C02566=1038.744,142.402,-96.604,169.943,40.243,157.587
C02567=1038.738,142.153,-96.582,169.941,40.243,157.587
C02568=1038.732,141.904,-96.561,169.939,40.243,157.587
C02569=1038.726,141.655,-96.539,169.937,40.242,157.587
C02570=1038.718,141.370,-96.515,169.934,40.242,157.586
C02571=1038.712,141.085,-96.490,169.932,40.242,157.586
C02572=1038.705,140.799,-96.465,169.928,40.241,157.586
C02573=1038.697,140.514,-96.441,169.926,40.241,157.586
C02574=1038.691,140.265,-96.419,169.924,40.240,157.586
C02575=1038.685,140.015,-96.398,169.921,40.240,157.586
C02576=1038.679,139.766,-96.376,169.919,40.240,157.585
C02577=1038.673,139.518,-96.355,169.917,40.239,157.585
C02578=1038.667,139.268,-96.333,169.915,40.239,157.585
C02579=1038.661,139.019,-96.312,169.912,40.239,157.585
C02580=1038.654,138.770,-96.291,169.910,40.239,157.585
C02581=1038.649,138.521,-96.270,169.907,40.238,157.585
C02582=1038.643,138.272,-96.248,169.905,40.238,157.585
C02583=1038.637,138.023,-96.226,169.903,40.238,157.584
C02584=1038.630,137.774,-96.205,169.901,40.238,157.584
C02585=1038.624,137.525,-96.184,169.898,40.237,157.584
C02586=1038.618,137.276,-96.163,169.896,40.237,157.584
C02587=1038.612,137.026,-96.142,169.893,40.237,157.584
C02588=1038.606,136.778,-96.121,169.891,40.237,157.584
C02589=1038.600,136.529,-96.099,169.889,40.236,157.583
C02590=1038.593,136.280,-96.078,169.887,40.236,157.583
C02591=1038.587,136.031,-96.057,169.885,40.236,157.583
C02592=1038.581,135.782,-96.036,169.883,40.235,157.583
C02593=1038.575,135.533,-96.014,169.879,40.235,157.583
C02594=1038.568,135.284,-95.993,169.877,40.235,157.583
C02595=1038.563,135.035,-95.972,169.875,40.235,157.583
C02596=1038.557,134.786,-95.950,169.873,40.234,157.582
C02597=1038.550,134.536,-95.930,169.871,40.234,157.582
C02598=1038.544,134.288,-95.909,169.869,40.234,157.582
C02599=1038.538,134.039,-95.887,169.866,40.234,157.582
C02600=1038.531,133.790,-95.866,169.864,40.233,157.582
C02601=1038.526,133.541,-95.846,169.861,40.233,157.582
C02602=1038.520,133.291,-95.824,169.859,40.233,157.581
C02603=1038.513,133.043,-95.803,169.857,40.233,157.581
C02604=1038.508,132.793,-95.782,169.855,40.232,157.581
C02605=1038.501,132.545,-95.761,169.853,40.232,157.581
C02606=1038.495,132.296,-95.740,169.850,40.231,157.581
C02607=1038.489,132.046,-95.719,169.848,40.232,157.581
C02608=1038.483,131.797,-95.698,169.845,40.231,157.581
C02609=1038.477,131.549,-95.677,169.843,40.231,157.580
C02610=1038.471,131.299,-95.656,169.841,40.230,157.580
C02611=1038.464,131.050,-95.635,169.839,40.231,157.580
C02612=1038.459,130.801,-95.614,169.837,40.230,157.580
C02613=1038.452,130.552,-95.593,169.835,40.230,157.580
C02614=1038.445,130.303,-95.572,169.832,40.230,157.580
C02615=1038.440,130.054,-95.552,169.830,40.230,157.580
C02616=1038.433,129.805,-95.531,169.828,40.230,157.580
C02617=1038.427,129.555,-95.510,169.825,40.229,157.579
C02618=1038.421,129.307,-95.489,169.823,40.229,157.579
C02619=1038.414,129.058,-95.469,169.821,40.229,157.579
C02620=1038.409,128.809,-95.448,169.818,40.229,157.579
C02621=1038.402,128.560,-95.427,169.816,40.229,157.579
C02622=1038.395,128.310,-95.407,169.814,40.228,157.579
C02623=1038.390,128.062,-95.386,169.812,40.229,157.579
C02624=1038.383,127.812,-95.365,169.810,40.228,157.579
C02625=1038.376,127.563,-95.344,169.808,40.228,157.578
C02626=1038.371,127.314,-95.324,169.805,40.228,157.578
C02627=1038.364,127.065,-95.303,169.802,40.228,157.578
C02628=1038.358,126.816,-95.283,169.800,40.228,157.578
C02629=1038.351,126.567,-95.262,169.798,40.227,157.578
C02630=1038.346,126.318,-95.241,169.796,40.227,157.578
C02631=1038.340,126.069,-95.221,169.794,40.227,157.578
C02632=1038.333,125.820,-95.200,169.792,40.227,157.577
C02633=1038.327,125.571,-95.179,169.790,40.226,157.577
C02634=1038.320,125.285,-95.155,169.787,40.227,157.577
C02635=1038.313,124.999,-95.131,169.784,40.226,157.577
C02636=1038.306,124.714,-95.108,169.781,40.226,157.577
C02637=1038.299,124.428,-95.085,169.779,40.226,157.577
C02638=1038.292,124.179,-95.064,169.777,40.226,157.577
C02639=1038.286,123.929,-95.044,169.775,40.225,157.576
C02640=1038.280,123.680,-95.023,169.773,40.225,157.576
C02641=1038.273,123.431,-95.002,169.770,40.225,157.576
C02642=1038.267,123.183,-94.982,169.768,40.225,157.576
C02643=1038.262,122.933,-94.961,169.766,40.225,157.576
C02644=1038.255,122.685,-94.940,169.763,40.224,157.576
C02645=1038.249,122.435,-94.920,169.761,40.224,157.576
C02646=1038.243,122.186,-94.900,169.759,40.224,157.576
C02647=1038.237,121.936,-94.879,169.757,40.224,157.575
C02648=1038.230,121.688,-94.859,169.755,40.224,157.575
C02649=1038.224,121.439,-94.838,169.753,40.223,157.575
C02650=1038.219,121.190,-94.818,169.751,40.224,157.575
C02651=1038.212,120.940,-94.797,169.748,40.223,157.575
C02652=1038.206,120.692,-94.777,169.745,40.223,157.575
C02653=1038.200,120.443,-94.756,169.743,40.223,157.575
C02654=1038.194,120.193,-94.736,169.741,40.223,157.575
C02655=1038.188,119.944,-94.716,169.739,40.222,157.574
C02656=1038.181,119.696,-94.695,169.737,40.222,157.574
C02657=1038.176,119.446,-94.674,169.735,40.222,157.574
C02658=1038.169,119.197,-94.654,169.733,40.222,157.574
C02659=1038.163,118.948,-94.634,169.731,40.222,157.574
C02660=1038.157,118.698,-94.613,169.729,40.221,157.574
C02661=1038.151,118.450,-94.593,169.727,40.221,157.574
C02662=1038.145,118.201,-94.572,169.724,40.221,157.573
C02663=1038.138,117.952,-94.552,169.722,40.220,157.573
C02664=1038.133,117.703,-94.531,169.720,40.221,157.573
C02665=1038.127,117.453,-94.511,169.717,40.220,157.573
C02666=1038.121,117.204,-94.491,169.715,40.220,157.573
C02667=1038.115,116.956,-94.471,169.713,40.220,157.573
C02668=1038.109,116.706,-94.450,169.711,40.220,157.573
C02669=1038.103,116.457,-94.430,169.708,40.219,157.572
C02670=1038.096,116.208,-94.409,169.706,40.219,157.572
C02671=1038.091,115.959,-94.389,169.704,40.219,157.572
C02672=1038.085,115.710,-94.369,169.702,40.218,157.572
C02673=1038.078,115.461,-94.348,169.700,40.219,157.572
C02674=1038.072,115.212,-94.329,169.698,40.218,157.572
C02675=1038.067,114.963,-94.308,169.696,40.218,157.572
C02676=1038.060,114.713,-94.288,169.694,40.218,157.572
C02677=1038.054,114.464,-94.268,169.692,40.218,157.571
C02678=1038.048,114.215,-94.248,169.689,40.217,157.571
C02679=1038.042,113.966,-94.227,169.687,40.217,157.571
C02680=1038.036,113.717,-94.207,169.685,40.217,157.571
C02681=1038.030,113.468,-94.187,169.683,40.216,157.571
C02682=1038.024,113.219,-94.167,169.681,40.217,157.571
C02683=1038.018,112.970,-94.147,169.679,40.216,157.571
C02684=1038.012,112.721,-94.127,169.676,40.216,157.571
C02685=1038.005,112.471,-94.106,169.674,40.216,157.570
C02686=1037.999,112.223,-94.086,169.672,40.216,157.570
C02687=1037.993,111.973,-94.066,169.669,40.216,157.570
C02688=1037.987,111.724,-94.046,169.667,40.216,157.570
C02689=1037.981,111.475,-94.027,169.665,40.216,157.570
C02690=1037.974,111.225,-94.006,169.663,40.216,157.570
C02691=1037.968,110.976,-93.987,169.661,40.215,157.570
C02692=1037.962,110.728,-93.967,169.659,40.215,157.570
C02693=1037.956,110.478,-93.946,169.657,40.215,157.570
C02694=1037.950,110.229,-93.926,169.655,40.215,157.569
C02695=1037.944,109.980,-93.907,169.653,40.215,157.569
C02696=1037.937,109.730,-93.887,169.651,40.215,157.569
C02697=1037.931,109.482,-93.867,169.649,40.215,157.569
C02698=1037.924,109.196,-93.844,169.646,40.215,157.569
C02699=1037.917,108.910,-93.822,169.643,40.214,157.569
C02700=1037.910,108.624,-93.799,169.640,40.215,157.569
C02701=1037.902,108.338,-93.776,169.638,40.214,157.569
C02702=1037.896,108.089,-93.756,169.636,40.214,157.569
C02703=1037.890,107.840,-93.737,169.634,40.214,157.568
C02704=1037.884,107.591,-93.717,169.632,40.214,157.568
C02705=1037.878,107.341,-93.697,169.630,40.214,157.568
C02706=1037.872,107.092,-93.677,169.628,40.214,157.568
C02707=1037.865,106.844,-93.658,169.626,40.213,157.568
C02708=1037.858,106.594,-93.638,169.624,40.214,157.568
C02709=1037.853,106.345,-93.618,169.621,40.213,157.568
C02710=1037.847,106.096,-93.598,169.619,40.213,157.568
C02711=1037.841,105.847,-93.579,169.617,40.213,157.567
C02712=1037.833,105.597,-93.559,169.614,40.213,157.567
C02713=1037.827,105.349,-93.539,169.612,40.213,157.567
C02714=1037.822,105.099,-93.520,169.610,40.213,157.567
C02715=1037.815,104.850,-93.500,169.608,40.213,157.567
C02716=1037.809,104.601,-93.480,169.606,40.213,157.567
C02717=1037.803,104.352,-93.461,169.604,40.212,157.567
C02718=1037.797,104.103,-93.441,169.602,40.213,157.567
C02719=1037.791,103.854,-93.421,169.599,40.212,157.567
C02720=1037.785,103.604,-93.401,169.597,40.212,157.566
C02721=1037.779,103.355,-93.382,169.595,40.212,157.566
C02722=1037.772,103.106,-93.363,169.593,40.212,157.566
C02723=1037.766,102.857,-93.343,169.591,40.212,157.566
C02724=1037.760,102.608,-93.323,169.589,40.212,157.566
C02725=1037.754,102.358,-93.303,169.587,40.211,157.566
C02726=1037.748,102.109,-93.283,169.585,40.212,157.566
C02727=1037.741,101.860,-93.265,169.583,40.211,157.566
C02728=1037.735,101.612,-93.245,169.581,40.211,157.566
C02729=1037.729,101.361,-93.225,169.579,40.211,157.565
C02730=1037.723,101.113,-93.205,169.577,40.211,157.565
C02731=1037.717,100.863,-93.187,169.574,40.211,157.565
C02732=1037.711,100.615,-93.167,169.572,40.211,157.565
C02733=1037.705,100.366,-93.147,169.570,40.210,157.565
C02734=1037.699,100.116,-93.127,169.568,40.211,157.565
C02735=1037.692,99.867,-93.108,169.566,40.210,157.565
C02736=1037.686,99.618,-93.088,169.564,40.210,157.565
C02737=1037.680,99.369,-93.070,169.562,40.210,157.564
C02738=1037.674,99.120,-93.050,169.559,40.210,157.564
C02739=1037.667,98.871,-93.031,169.557,40.210,157.564
C02740=1037.661,98.621,-93.011,169.555,40.210,157.564
C02741=1037.654,98.372,-92.992,169.553,40.210,157.564
C02742=1037.648,98.123,-92.973,169.551,40.210,157.564
C02743=1037.642,97.874,-92.954,169.548,40.210,157.564
C02744=1037.636,97.625,-92.934,169.546,40.210,157.564
C02745=1037.629,97.375,-92.915,169.544,40.210,157.564
C02746=1037.623,97.126,-92.895,169.542,40.210,157.564
C02747=1037.617,96.877,-92.877,169.540,40.210,157.564
C02748=1037.611,96.628,-92.857,169.538,40.210,157.563
C02749=1037.605,96.379,-92.838,169.536,40.210,157.563
C02750=1037.598,96.130,-92.819,169.534,40.209,157.563
C02751=1037.593,95.880,-92.800,169.532,40.209,157.563
C02752=1037.585,95.631,-92.780,169.530,40.210,157.563
C02753=1037.580,95.382,-92.761,169.528,40.209,157.563
C02754=1037.573,95.132,-92.742,169.526,40.209,157.563
C02755=1037.567,94.884,-92.722,169.523,40.209,157.563
C02756=1037.561,94.634,-92.703,169.521,40.209,157.563
C02757=1037.555,94.385,-92.684,169.519,40.209,157.562
C02758=1037.549,94.136,-92.665,169.517,40.209,157.562
C02759=1037.543,93.887,-92.646,169.515,40.209,157.562
C02760=1037.536,93.637,-92.627,169.513,40.209,157.562
C02761=1037.530,93.388,-92.607,169.511,40.209,157.562
C02762=1037.523,93.103,-92.585,169.508,40.209,157.562
C02763=1037.516,92.817,-92.564,169.506,40.209,157.562
C02764=1037.509,92.531,-92.541,169.504,40.208,157.562
C02765=1037.502,92.244,-92.520,169.501,40.209,157.562
C02766=1037.495,91.995,-92.501,169.498,40.208,157.561
C02767=1037.489,91.747,-92.481,169.496,40.208,157.561
C02768=1037.483,91.497,-92.462,169.494,40.208,157.561
C02769=1037.477,91.248,-92.443,169.492,40.208,157.561
C02770=1037.471,90.999,-92.425,169.490,40.208,157.561
C02771=1037.465,90.749,-92.405,169.488,40.208,157.561
C02772=1037.458,90.500,-92.387,169.486,40.208,157.561
C02773=1037.452,90.252,-92.367,169.484,40.208,157.561
C02774=1037.446,90.002,-92.348,169.482,40.208,157.561
C02775=1037.440,89.753,-92.329,169.480,40.207,157.561
C02776=1037.434,89.504,-92.310,169.478,40.207,157.560
C02777=1037.427,89.254,-92.291,169.476,40.208,157.560
C02778=1037.420,89.005,-92.272,169.473,40.207,157.560
C02779=1037.414,88.756,-92.254,169.471,40.207,157.560
C02780=1037.408,88.506,-92.235,169.469,40.208,157.560
C02781=1037.402,88.257,-92.216,169.467,40.208,157.560
C02782=1037.396,88.008,-92.197,169.465,40.207,157.560
C02783=1037.389,87.759,-92.179,169.463,40.208,157.560
C02784=1037.383,87.510,-92.160,169.461,40.208,157.560
C02785=1037.377,87.260,-92.141,169.459,40.207,157.560
C02786=1037.371,87.011,-92.122,169.457,40.208,157.560
C02787=1037.364,86.762,-92.103,169.455,40.208,157.560
C02788=1037.358,86.513,-92.085,169.453,40.207,157.559
C02789=1037.351,86.264,-92.066,169.451,40.207,157.559
C02790=1037.346,86.014,-92.047,169.449,40.208,157.559
C02791=1037.339,85.765,-92.028,169.447,40.207,157.559
C02792=1037.333,85.516,-92.010,169.444,40.207,157.559
C02793=1037.326,85.267,-91.991,169.442,40.208,157.559
C02794=1037.320,85.018,-91.972,169.439,40.207,157.559
C02795=1037.314,84.769,-91.953,169.437,40.207,157.559
C02796=1037.308,84.519,-91.934,169.435,40.208,157.559
C02797=1037.301,84.270,-91.916,169.433,40.207,157.559
C02798=1037.295,84.021,-91.897,169.431,40.207,157.559
C02799=1037.289,83.771,-91.879,169.429,40.208,157.558
C02800=1037.283,83.522,-91.860,169.427,40.207,157.558
C02801=1037.277,83.273,-91.841,169.425,40.207,157.558
C02802=1037.270,83.024,-91.823,169.423,40.208,157.558
C02803=1037.264,82.775,-91.804,169.421,40.207,157.558
C02804=1037.257,82.526,-91.785,169.419,40.207,157.558
C02805=1037.251,82.276,-91.767,169.417,40.207,157.558
C02806=1037.245,82.027,-91.747,169.415,40.207,157.558
C02807=1037.239,81.777,-91.730,169.413,40.207,157.558
C02808=1037.233,81.528,-91.711,169.410,40.207,157.558
C02809=1037.226,81.279,-91.692,169.408,40.207,157.557
C02810=1037.220,81.031,-91.674,169.406,40.207,157.557
C02811=1037.214,80.781,-91.655,169.404,40.207,157.557
C02812=1037.208,80.532,-91.636,169.402,40.207,157.557
C02813=1037.202,80.282,-91.618,169.400,40.207,157.557
C02814=1037.196,80.033,-91.599,169.398,40.207,157.557
C02815=1037.189,79.784,-91.581,169.396,40.207,157.557
C02816=1037.183,79.535,-91.562,169.394,40.206,157.557
C02817=1037.177,79.285,-91.544,169.392,40.207,157.557
C02818=1037.171,79.036,-91.525,169.390,40.207,157.557
C02819=1037.165,78.787,-91.506,169.388,40.206,157.556
C02820=1037.159,78.538,-91.488,169.386,40.206,157.556
C02821=1037.153,78.288,-91.470,169.383,40.206,157.556
C02822=1037.146,78.039,-91.451,169.381,40.206,157.556
C02823=1037.140,77.790,-91.433,169.379,40.206,157.556
C02824=1037.134,77.541,-91.414,169.377,40.207,157.556
C02825=1037.127,77.291,-91.396,169.375,40.206,157.556
C02826=1037.118,76.901,-91.367,169.372,40.206,157.556
C02827=1037.108,76.512,-91.339,169.369,40.206,157.556
C02828=1037.098,76.122,-91.310,169.365,40.207,157.556
C02829=1037.088,75.733,-91.282,169.362,40.206,157.555
C02830=1037.081,75.484,-91.263,169.360,40.206,157.555
C02831=1037.076,75.235,-91.245,169.358,40.207,157.555
C02832=1037.070,74.985,-91.227,169.356,40.207,157.555
C02833=1037.063,74.736,-91.208,169.353,40.206,157.555
C02834=1037.057,74.487,-91.190,169.351,40.206,157.555
C02835=1037.051,74.237,-91.172,169.349,40.207,157.555
C02836=1037.044,73.988,-91.154,169.347,40.207,157.555
C02837=1037.037,73.739,-91.136,169.345,40.206,157.555
C02838=1037.032,73.490,-91.118,169.343,40.207,157.555
C02839=1037.025,73.241,-91.100,169.341,40.207,157.555
C02840=1037.019,72.992,-91.081,169.339,40.206,157.554
C02841=1037.013,72.742,-91.063,169.337,40.207,157.554
C02842=1037.006,72.493,-91.044,169.335,40.207,157.554
C02843=1037.001,72.244,-91.027,169.333,40.206,157.554
C02844=1036.994,71.995,-91.008,169.331,40.206,157.554
C02845=1036.988,71.745,-90.990,169.329,40.207,157.554
C02846=1036.981,71.496,-90.972,169.327,40.207,157.554
C02847=1036.975,71.246,-90.954,169.325,40.206,157.554
C02848=1036.969,70.997,-90.936,169.323,40.207,157.554
C02849=1036.963,70.748,-90.918,169.321,40.207,157.554
C02850=1036.957,70.498,-90.900,169.318,40.206,157.554
C02851=1036.951,70.249,-90.881,169.316,40.207,157.554
C02852=1036.944,70.000,-90.864,169.314,40.207,157.553
C02853=1036.938,69.751,-90.846,169.312,40.207,157.553
C02854=1036.932,69.502,-90.828,169.310,40.206,157.553
C02855=1036.926,69.252,-90.810,169.308,40.207,157.553
C02856=1036.919,69.003,-90.791,169.305,40.207,157.553
C02857=1036.912,68.753,-90.774,169.303,40.207,157.553
C02858=1036.906,68.505,-90.756,169.301,40.207,157.553
C02859=1036.900,68.255,-90.738,169.299,40.207,157.553
C02860=1036.894,68.005,-90.720,169.297,40.207,157.553
C02861=1036.887,67.757,-90.702,169.295,40.207,157.553
C02862=1036.882,67.508,-90.684,169.293,40.207,157.553
C02863=1036.875,67.258,-90.666,169.291,40.207,157.553
C02864=1036.868,67.009,-90.648,169.289,40.207,157.553
C02865=1036.862,66.759,-90.630,169.286,40.207,157.552
C02866=1036.857,66.510,-90.613,169.284,40.207,157.552
C02867=1036.850,66.261,-90.594,169.282,40.207,157.552
C02868=1036.843,66.012,-90.577,169.280,40.207,157.552
C02869=1036.837,65.762,-90.559,169.278,40.208,157.552
C02870=1036.831,65.513,-90.542,169.276,40.207,157.552
C02871=1036.825,65.264,-90.523,169.274,40.207,157.552
C02872=1036.818,65.014,-90.505,169.272,40.208,157.552
C02873=1036.812,64.765,-90.488,169.270,40.208,157.552
C02874=1036.806,64.516,-90.470,169.268,40.207,157.552
C02875=1036.800,64.267,-90.452,169.266,40.207,157.552
C02876=1036.793,64.017,-90.434,169.264,40.208,157.552
C02877=1036.787,63.768,-90.417,169.262,40.208,157.551
C02878=1036.777,63.373,-90.389,169.258,40.208,157.551
C02879=1036.767,62.978,-90.362,169.255,40.208,157.551
C02880=1036.756,62.583,-90.333,169.252,40.208,157.551
C02881=1036.746,62.188,-90.305,169.249,40.208,157.551
C02882=1036.739,61.939,-90.288,169.246,40.209,157.551
C02883=1036.733,61.689,-90.270,169.244,40.209,157.551
C02884=1036.727,61.440,-90.253,169.242,40.209,157.551
C02885=1036.720,61.191,-90.236,169.240,40.209,157.551
C02886=1036.713,60.904,-90.215,169.237,40.209,157.551
C02887=1036.706,60.618,-90.195,169.234,40.209,157.551
C02888=1036.698,60.332,-90.175,169.232,40.209,157.551
C02889=1036.691,60.046,-90.155,169.230,40.210,157.550
C02890=1036.684,59.796,-90.138,169.228,40.210,157.550
C02891=1036.679,59.547,-90.120,169.226,40.210,157.550
C02892=1036.672,59.298,-90.103,169.223,40.210,157.550
C02893=1036.665,59.049,-90.085,169.221,40.210,157.550
C02894=1036.660,58.800,-90.068,169.219,40.210,157.550
C02895=1036.653,58.550,-90.051,169.217,40.210,157.550
C02896=1036.646,58.301,-90.033,169.215,40.210,157.550
C02897=1036.640,58.052,-90.016,169.213,40.211,157.550
C02898=1036.633,57.802,-89.998,169.211,40.211,157.550
C02899=1036.627,57.553,-89.981,169.209,40.211,157.550
C02900=1036.621,57.304,-89.963,169.207,40.211,157.550
C02901=1036.614,57.054,-89.946,169.205,40.211,157.550
C02902=1036.608,56.805,-89.928,169.203,40.211,157.550
C02903=1036.602,56.556,-89.911,169.201,40.211,157.550
C02904=1036.595,56.306,-89.894,169.199,40.211,157.549
C02905=1036.589,56.057,-89.876,169.197,40.211,157.549
C02906=1036.583,55.808,-89.859,169.194,40.212,157.549
C02907=1036.576,55.558,-89.842,169.192,40.212,157.549
C02908=1036.570,55.309,-89.824,169.189,40.211,157.549
C02909=1036.563,55.060,-89.807,169.187,40.212,157.549
C02910=1036.557,54.811,-89.790,169.185,40.212,157.549
C02911=1036.551,54.561,-89.772,169.183,40.212,157.549
C02912=1036.544,54.311,-89.755,169.181,40.212,157.549
C02913=1036.538,54.063,-89.738,169.179,40.212,157.549
C02914=1036.532,53.813,-89.720,169.177,40.212,157.549
C02915=1036.526,53.564,-89.703,169.175,40.212,157.549
C02916=1036.519,53.315,-89.686,169.173,40.212,157.549
C02917=1036.513,53.066,-89.668,169.171,40.213,157.549
C02918=1036.507,52.816,-89.652,169.169,40.213,157.549
C02919=1036.500,52.566,-89.634,169.167,40.212,157.548
C02920=1036.495,52.317,-89.617,169.165,40.213,157.548
C02921=1036.488,52.068,-89.599,169.163,40.213,157.548
C02922=1036.481,51.819,-89.582,169.161,40.213,157.548
C02923=1036.476,51.569,-89.565,169.158,40.213,157.548
C02924=1036.469,51.320,-89.548,169.156,40.213,157.548
C02925=1036.462,51.071,-89.531,169.154,40.213,157.548
C02926=1036.457,50.822,-89.513,169.152,40.213,157.548
C02927=1036.450,50.572,-89.496,169.150,40.213,157.548
C02928=1036.444,50.323,-89.480,169.148,40.214,157.548
C02929=1036.437,50.073,-89.462,169.145,40.213,157.548
C02930=1036.432,49.824,-89.445,169.143,40.213,157.548
C02931=1036.425,49.575,-89.428,169.141,40.213,157.547
C02932=1036.419,49.326,-89.411,169.139,40.214,157.547
C02933=1036.413,49.076,-89.393,169.137,40.214,157.547
C02934=1036.407,48.827,-89.376,169.135,40.213,157.547
C02935=1036.400,48.578,-89.359,169.133,40.214,157.547
C02936=1036.395,48.328,-89.342,169.131,40.214,157.547
C02937=1036.388,48.079,-89.325,169.129,40.214,157.547
C02938=1036.381,47.830,-89.308,169.127,40.214,157.547
C02939=1036.375,47.580,-89.291,169.125,40.214,157.547
C02940=1036.369,47.331,-89.274,169.123,40.214,157.547
C02941=1036.362,47.081,-89.256,169.120,40.214,157.547
C02942=1036.357,46.832,-89.240,169.118,40.214,157.547
C02943=1036.351,46.583,-89.223,169.116,40.214,157.546
C02944=1036.344,46.333,-89.205,169.114,40.214,157.546
C02945=1036.338,46.084,-89.189,169.112,40.214,157.546
C02946=1036.332,45.834,-89.171,169.110,40.215,157.546
C02947=1036.326,45.586,-89.154,169.107,40.214,157.546
C02948=1036.320,45.336,-89.138,169.105,40.214,157.546
C02949=1036.313,45.087,-89.120,169.103,40.214,157.546
C02950=1036.306,44.800,-89.101,169.101,40.215,157.546
C02951=1036.299,44.514,-89.081,169.098,40.214,157.546
C02952=1036.292,44.227,-89.062,169.096,40.214,157.546
C02953=1036.285,43.941,-89.042,169.094,40.215,157.546
C02954=1036.279,43.691,-89.025,169.092,40.214,157.546
C02955=1036.273,43.442,-89.009,169.090,40.214,157.545
C02956=1036.267,43.193,-88.991,169.088,40.215,157.545
C02957=1036.261,42.943,-88.975,169.085,40.215,157.545
C02958=1036.254,42.694,-88.958,169.083,40.215,157.545
C02959=1036.248,42.444,-88.941,169.081,40.215,157.545
C02960=1036.242,42.195,-88.924,169.079,40.215,157.545
C02961=1036.236,41.946,-88.908,169.077,40.215,157.545
C02962=1036.229,41.696,-88.890,169.075,40.215,157.545
C02963=1036.223,41.447,-88.874,169.073,40.215,157.545
C02964=1036.216,41.198,-88.857,169.071,40.216,157.545
C02965=1036.210,40.948,-88.841,169.069,40.216,157.545
C02966=1036.204,40.700,-88.824,169.067,40.216,157.545
C02967=1036.197,40.450,-88.807,169.065,40.216,157.545
C02968=1036.191,40.200,-88.791,169.061,40.216,157.545
C02969=1036.185,39.951,-88.774,169.059,40.216,157.544
C02970=1036.178,39.701,-88.757,169.057,40.216,157.544
C02971=1036.172,39.453,-88.740,169.055,40.216,157.544
C02972=1036.166,39.203,-88.724,169.053,40.217,157.544
C02973=1036.160,38.953,-88.707,169.051,40.217,157.544
C02974=1036.153,38.705,-88.690,169.049,40.217,157.544
C02975=1036.147,38.454,-88.674,169.047,40.217,157.544
C02976=1036.141,38.205,-88.657,169.045,40.217,157.544
C02977=1036.135,37.956,-88.641,169.043,40.217,157.544
C02978=1036.128,37.706,-88.624,169.041,40.217,157.544
C02979=1036.122,37.457,-88.608,169.038,40.217,157.544
C02980=1036.116,37.208,-88.591,169.036,40.218,157.544
C02981=1036.109,36.958,-88.574,169.034,40.218,157.544
C02982=1036.103,36.709,-88.558,169.032,40.218,157.544
C02983=1036.097,36.460,-88.542,169.030,40.218,157.544
C02984=1036.090,36.210,-88.525,169.028,40.218,157.543
C02985=1036.084,35.961,-88.509,169.026,40.218,157.543
C02986=1036.078,35.712,-88.492,169.024,40.218,157.543
C02987=1036.071,35.462,-88.476,169.021,40.218,157.543
C02988=1036.065,35.213,-88.460,169.019,40.219,157.543
C02989=1036.058,34.964,-88.443,169.017,40.219,157.543
C02990=1036.052,34.714,-88.426,169.015,40.219,157.543
C02991=1036.046,34.465,-88.410,169.013,40.219,157.543
C02992=1036.039,34.215,-88.394,169.011,40.219,157.543
C02993=1036.033,33.965,-88.378,169.009,40.220,157.543
C02994=1036.026,33.717,-88.361,169.006,40.220,157.543
C02995=1036.020,33.467,-88.345,169.003,40.220,157.543
C02996=1036.014,33.218,-88.329,169.001,40.220,157.543
C02997=1036.007,32.968,-88.312,168.999,40.220,157.543
C02998=1036.001,32.719,-88.296,168.997,40.221,157.543
C02999=1035.995,32.470,-88.280,168.995,40.221,157.543
C03000=1035.989,32.219,-88.263,168.993,40.221,157.543
C03001=1035.982,31.971,-88.247,168.991,40.221,157.543
C03002=1035.976,31.722,-88.231,168.989,40.221,157.543
C03003=1035.970,31.472,-88.214,168.986,40.221,157.542
C03004=1035.963,31.222,-88.198,168.984,40.221,157.542
C03005=1035.957,30.973,-88.182,168.982,40.221,157.542
C03006=1035.951,30.724,-88.166,168.980,40.222,157.542
C03007=1035.945,30.475,-88.150,168.978,40.222,157.542
C03008=1035.939,30.225,-88.133,168.976,40.222,157.542
C03009=1035.931,29.976,-88.117,168.974,40.222,157.542
C03010=1035.926,29.726,-88.101,168.971,40.222,157.542
C03011=1035.920,29.477,-88.085,168.969,40.223,157.542
C03012=1035.914,29.227,-88.068,168.967,40.223,157.542
C03013=1035.906,28.978,-88.052,168.965,40.223,157.542
C03014=1035.900,28.691,-88.033,168.963,40.223,157.542
C03015=1035.892,28.405,-88.015,168.960,40.223,157.542
C03016=1035.885,28.119,-87.996,168.958,40.223,157.542
C03017=1035.878,27.832,-87.978,168.955,40.223,157.541
C03018=1035.872,27.582,-87.962,168.953,40.224,157.541
C03019=1035.865,27.333,-87.946,168.951,40.224,157.541
C03020=1035.859,27.083,-87.929,168.949,40.224,157.541
C03021=1035.852,26.834,-87.914,168.947,40.224,157.541
C03022=1035.846,26.585,-87.898,168.945,40.224,157.541
C03023=1035.839,26.336,-87.882,168.941,40.225,157.541
C03024=1035.833,26.087,-87.866,168.939,40.225,157.541
C03025=1035.827,25.837,-87.849,168.937,40.225,157.541
C03026=1035.820,25.587,-87.834,168.935,40.225,157.541
C03027=1035.814,25.338,-87.818,168.933,40.225,157.541
C03028=1035.808,25.089,-87.802,168.931,40.226,157.541
C03029=1035.802,24.839,-87.786,168.928,40.226,157.541
C03030=1035.795,24.590,-87.770,168.926,40.226,157.541
C03031=1035.789,24.340,-87.754,168.924,40.226,157.541
C03032=1035.782,24.091,-87.738,168.922,40.226,157.541
C03033=1035.776,23.841,-87.722,168.920,40.227,157.541
C03034=1035.770,23.592,-87.707,168.918,40.227,157.541
C03035=1035.764,23.343,-87.690,168.915,40.227,157.540
C03036=1035.757,23.094,-87.675,168.913,40.227,157.540
C03037=1035.751,22.844,-87.659,168.911,40.228,157.540
C03038=1035.744,22.594,-87.643,168.909,40.228,157.540
C03039=1035.738,22.345,-87.627,168.907,40.228,157.540
C03040=1035.731,22.096,-87.611,168.904,40.228,157.540
C03041=1035.725,21.846,-87.595,168.902,40.228,157.540
C03042=1035.719,21.597,-87.580,168.900,40.229,157.540
C03043=1035.713,21.347,-87.564,168.898,40.229,157.540
C03044=1035.706,21.098,-87.548,168.896,40.229,157.540
C03045=1035.700,20.849,-87.532,168.894,40.229,157.540
C03046=1035.694,20.599,-87.517,168.891,40.229,157.540
C03047=1035.687,20.349,-87.500,168.889,40.230,157.540
C03048=1035.681,20.100,-87.485,168.887,40.230,157.540
C03049=1035.675,19.851,-87.468,168.885,40.230,157.540
C03050=1035.668,19.601,-87.453,168.883,40.230,157.540
C03051=1035.662,19.352,-87.437,168.881,40.230,157.540
C03052=1035.656,19.103,-87.422,168.878,40.231,157.540
C03053=1035.649,18.853,-87.407,168.876,40.231,157.540
C03054=1035.643,18.604,-87.390,168.874,40.231,157.539
C03055=1035.637,18.354,-87.375,168.872,40.231,157.539
C03056=1035.630,18.105,-87.360,168.870,40.232,157.539
C03057=1035.624,17.856,-87.344,168.867,40.232,157.539
C03058=1035.618,17.606,-87.329,168.865,40.233,157.539
C03059=1035.611,17.357,-87.313,168.863,40.233,157.539
C03060=1035.606,17.107,-87.297,168.861,40.233,157.539
C03061=1035.598,16.857,-87.281,168.859,40.233,157.539
C03062=1035.592,16.608,-87.265,168.856,40.234,157.539
C03063=1035.586,16.358,-87.250,168.854,40.234,157.539
C03064=1035.579,16.109,-87.234,168.852,40.234,157.539
C03065=1035.574,15.859,-87.219,168.850,40.234,157.539
C03066=1035.567,15.610,-87.203,168.848,40.234,157.539
C03067=1035.561,15.361,-87.188,168.845,40.235,157.539
C03068=1035.555,15.111,-87.172,168.843,40.235,157.539
C03069=1035.548,14.862,-87.156,168.841,40.235,157.539
C03070=1035.542,14.612,-87.141,168.838,40.235,157.539
C03071=1035.536,14.363,-87.126,168.836,40.235,157.539
C03072=1035.529,14.113,-87.110,168.833,40.236,157.539
C03073=1035.523,13.864,-87.095,168.831,40.236,157.539
C03074=1035.516,13.615,-87.080,168.829,40.236,157.538
C03075=1035.510,13.365,-87.065,168.827,40.236,157.538
C03076=1035.504,13.116,-87.048,168.824,40.237,157.538
C03077=1035.498,12.866,-87.033,168.822,40.237,157.538
C03078=1035.490,12.581,-87.016,168.820,40.238,157.538
C03079=1035.482,12.296,-86.998,168.817,40.238,157.538
C03080=1035.475,12.010,-86.981,168.814,40.238,157.538
C03081=1035.468,11.725,-86.964,168.812,40.238,157.538
C03082=1035.462,11.476,-86.949,168.810,40.239,157.538
C03083=1035.455,11.227,-86.933,168.807,40.239,157.538
C03084=1035.449,10.977,-86.918,168.805,40.240,157.538
C03085=1035.442,10.728,-86.903,168.803,40.240,157.538
C03086=1035.436,10.478,-86.888,168.801,40.240,157.538
C03087=1035.429,10.229,-86.873,168.798,40.240,157.538
C03088=1035.423,9.979,-86.858,168.796,40.241,157.538
C03089=1035.416,9.730,-86.842,168.794,40.241,157.538
C03090=1035.410,9.480,-86.827,168.792,40.242,157.538
C03091=1035.404,9.231,-86.812,168.789,40.242,157.538
C03092=1035.398,8.981,-86.796,168.787,40.242,157.538
C03093=1035.391,8.732,-86.781,168.785,40.242,157.538
C03094=1035.385,8.482,-86.766,168.783,40.242,157.538
C03095=1035.378,8.233,-86.750,168.780,40.243,157.538
C03096=1035.372,7.983,-86.735,168.778,40.244,157.538
C03097=1035.365,7.734,-86.721,168.776,40.244,157.538
C03098=1035.359,7.484,-86.706,168.774,40.244,157.538
C03099=1035.353,7.234,-86.691,168.771,40.244,157.538
C03100=1035.347,6.986,-86.675,168.769,40.244,157.537
C03101=1035.340,6.736,-86.660,168.767,40.245,157.537
C03102=1035.334,6.487,-86.645,168.764,40.245,157.537
C03103=1035.327,6.237,-86.631,168.762,40.246,157.537
C03104=1035.321,5.988,-86.615,168.760,40.246,157.537
C03105=1035.314,5.738,-86.600,168.758,40.246,157.537
C03106=1035.308,5.489,-86.585,168.755,40.246,157.537
C03107=1035.302,5.239,-86.570,168.753,40.247,157.537
C03108=1035.296,4.990,-86.555,168.751,40.247,157.537
C03109=1035.289,4.740,-86.540,168.749,40.247,157.537
C03110=1035.283,4.491,-86.525,168.746,40.247,157.537
C03111=1035.276,4.242,-86.510,168.744,40.248,157.537
C03112=1035.270,3.992,-86.495,168.742,40.248,157.537
C03113=1035.264,3.742,-86.479,168.740,40.249,157.537
C03114=1035.258,3.492,-86.464,168.737,40.249,157.537
C03115=1035.252,3.243,-86.450,168.735,40.249,157.537
C03116=1035.246,2.994,-86.435,168.733,40.249,157.537
C03117=1035.239,2.744,-86.420,168.731,40.249,157.537
C03118=1035.233,2.495,-86.404,168.728,40.250,157.537
C03119=1035.226,2.245,-86.389,168.726,40.250,157.537
C03120=1035.220,1.996,-86.375,168.724,40.250,157.537
C03121=1035.214,1.747,-86.360,168.721,40.251,157.537
C03122=1035.208,1.497,-86.345,168.719,40.251,157.537
C03123=1035.201,1.248,-86.330,168.717,40.251,157.537
C03124=1035.195,0.998,-86.315,168.715,40.252,157.536
C03125=1035.189,0.749,-86.300,168.712,40.252,157.536
C03126=1035.183,0.499,-86.285,168.710,40.252,157.536
C03127=1035.176,0.250,-86.271,168.708,40.252,157.536
C03128=1035.170,-0.000,-86.256,168.706,40.253,157.536
C03129=1035.164,-0.249,-86.241,168.703,40.253,157.536
C03130=1035.158,-0.499,-86.226,168.701,40.253,157.536
C03131=1035.151,-0.748,-86.211,168.699,40.253,157.536
C03132=1035.145,-0.998,-86.196,168.696,40.254,157.536
C03133=1035.139,-1.247,-86.182,168.694,40.254,157.536
C03134=1035.133,-1.497,-86.167,168.692,40.255,157.536
C03135=1035.127,-1.746,-86.152,168.690,40.255,157.536
C03136=1035.120,-1.996,-86.137,168.687,40.255,157.536
C03137=1035.114,-2.245,-86.122,168.685,40.255,157.536
C03138=1035.108,-2.495,-86.107,168.683,40.255,157.536
C03139=1035.102,-2.744,-86.092,168.680,40.256,157.536
C03140=1035.096,-2.993,-86.078,168.678,40.256,157.536
C03141=1035.089,-3.243,-86.063,168.676,40.256,157.536
C03142=1035.082,-3.526,-86.046,168.673,40.256,157.536
C03143=1035.075,-3.810,-86.030,168.671,40.257,157.536
C03144=1035.068,-4.093,-86.014,168.668,40.258,157.536
C03145=1035.060,-4.377,-85.996,168.665,40.258,157.535
C03146=1035.055,-4.626,-85.982,168.663,40.258,157.535
C03147=1035.048,-4.876,-85.968,168.661,40.259,157.535
C03148=1035.041,-5.125,-85.953,168.658,40.259,157.535
C03149=1035.035,-5.374,-85.939,168.656,40.259,157.535
C03150=1035.028,-5.624,-85.924,168.654,40.260,157.535
C03151=1035.022,-5.874,-85.910,168.651,40.261,157.535
C03152=1035.016,-6.124,-85.895,168.649,40.261,157.535
C03153=1035.009,-6.372,-85.881,168.647,40.261,157.535
C03154=1035.003,-6.622,-85.866,168.644,40.261,157.535
C03155=1034.997,-6.872,-85.852,168.642,40.262,157.535
C03156=1034.990,-7.121,-85.838,168.640,40.262,157.535
C03157=1034.984,-7.370,-85.823,168.637,40.263,157.535
C03158=1034.978,-7.621,-85.809,168.635,40.263,157.535
C03159=1034.971,-7.869,-85.795,168.632,40.264,157.535
C03160=1034.965,-8.119,-85.780,168.630,40.264,157.535
C03161=1034.959,-8.369,-85.766,168.628,40.264,157.535
C03162=1034.952,-8.618,-85.752,168.625,40.264,157.535
C03163=1034.946,-8.868,-85.737,168.623,40.265,157.535
C03164=1034.940,-9.118,-85.722,168.621,40.265,157.535
C03165=1034.933,-9.367,-85.708,168.618,40.266,157.535
C03166=1034.927,-9.616,-85.693,168.616,40.266,157.535
C03167=1034.921,-9.866,-85.679,168.614,40.267,157.535
C03168=1034.914,-10.115,-85.665,168.611,40.267,157.535
C03169=1034.908,-10.365,-85.650,168.609,40.267,157.535
C03170=1034.902,-10.614,-85.637,168.607,40.267,157.535
C03171=1034.895,-10.864,-85.622,168.604,40.268,157.535
C03172=1034.889,-11.114,-85.608,168.602,40.269,157.535
C03173=1034.883,-11.363,-85.594,168.599,40.269,157.535
C03174=1034.876,-11.612,-85.579,168.597,40.269,157.535
C03175=1034.871,-11.862,-85.565,168.595,40.270,157.535
C03176=1034.864,-12.111,-85.551,168.592,40.270,157.535
C03177=1034.858,-12.361,-85.536,168.590,40.270,157.535
C03178=1034.851,-12.610,-85.522,168.588,40.271,157.535
C03179=1034.845,-12.860,-85.508,168.585,40.272,157.535
C03180=1034.839,-13.109,-85.494,168.583,40.272,157.535
C03181=1034.833,-13.359,-85.480,168.581,40.272,157.534
C03182=1034.827,-13.608,-85.465,168.578,40.272,157.534
C03183=1034.821,-13.859,-85.451,168.576,40.272,157.534
C03184=1034.814,-14.107,-85.437,168.573,40.273,157.534
C03185=1034.808,-14.357,-85.423,168.571,40.274,157.534
C03186=1034.802,-14.606,-85.409,168.569,40.274,157.534
C03187=1034.796,-14.856,-85.395,168.566,40.274,157.534
C03188=1034.789,-15.106,-85.380,168.564,40.275,157.534
C03189=1034.783,-15.355,-85.367,168.562,40.275,157.534
C03190=1034.777,-15.605,-85.352,168.559,40.275,157.534
C03191=1034.770,-15.854,-85.338,168.557,40.276,157.534
C03192=1034.763,-16.104,-85.324,168.554,40.277,157.534
C03193=1034.758,-16.353,-85.310,168.552,40.277,157.534
C03194=1034.751,-16.603,-85.296,168.549,40.278,157.534
C03195=1034.745,-16.852,-85.282,168.547,40.278,157.534
C03196=1034.738,-17.102,-85.268,168.545,40.278,157.534
C03197=1034.732,-17.351,-85.255,168.542,40.279,157.534
C03198=1034.726,-17.601,-85.240,168.540,40.279,157.534
C03199=1034.720,-17.850,-85.227,168.537,40.280,157.534
C03200=1034.713,-18.100,-85.213,168.535,40.280,157.534
C03201=1034.707,-18.349,-85.199,168.532,40.281,157.534
C03202=1034.700,-18.599,-85.185,168.531,40.282,157.534
C03203=1034.694,-18.848,-85.172,168.529,40.282,157.534
C03204=1034.688,-19.098,-85.157,168.525,40.282,157.534
C03205=1034.681,-19.347,-85.143,168.524,40.283,157.534
C03206=1034.674,-19.630,-85.128,168.521,40.283,157.534
C03207=1034.667,-19.911,-85.112,168.518,40.283,157.534
C03208=1034.660,-20.193,-85.096,168.516,40.284,157.534
C03209=1034.653,-20.474,-85.081,168.513,40.285,157.534
C03210=1034.646,-20.724,-85.068,168.510,40.286,157.534
C03211=1034.640,-20.973,-85.053,168.508,40.286,157.534
C03212=1034.634,-21.223,-85.039,168.505,40.286,157.534
C03213=1034.627,-21.473,-85.026,168.503,40.287,157.534
C03214=1034.621,-21.723,-85.012,168.501,40.287,157.534
C03215=1034.615,-21.972,-84.999,168.498,40.287,157.534
C03216=1034.608,-22.221,-84.984,168.496,40.288,157.534
C03217=1034.603,-22.471,-84.970,168.493,40.289,157.534
C03218=1034.596,-22.720,-84.957,168.491,40.289,157.534
C03219=1034.589,-22.970,-84.943,168.488,40.290,157.534
C03220=1034.584,-23.220,-84.930,168.486,40.290,157.534
C03221=1034.577,-23.470,-84.916,168.483,40.290,157.534
C03222=1034.571,-23.718,-84.902,168.481,40.291,157.534
C03223=1034.565,-23.968,-84.888,168.479,40.291,157.534
C03224=1034.558,-24.218,-84.874,168.476,40.291,157.533
C03225=1034.552,-24.467,-84.861,168.474,40.292,157.534
C03226=1034.547,-24.717,-84.847,168.471,40.293,157.533
C03227=1034.540,-24.967,-84.834,168.469,40.293,157.534
C03228=1034.534,-25.216,-84.820,168.466,40.294,157.533
C03229=1034.528,-25.466,-84.807,168.464,40.294,157.533
C03230=1034.521,-25.716,-84.793,168.461,40.295,157.533
C03231=1034.515,-25.965,-84.780,168.459,40.295,157.533
C03232=1034.510,-26.214,-84.766,168.457,40.295,157.533
C03233=1034.503,-26.464,-84.751,168.454,40.296,157.533
C03234=1034.496,-26.713,-84.738,168.452,40.296,157.533
C03235=1034.490,-26.963,-84.725,168.449,40.297,157.533
C03236=1034.484,-27.213,-84.711,168.447,40.298,157.533
C03237=1034.478,-27.462,-84.697,168.444,40.298,157.533
C03238=1034.471,-27.712,-84.684,168.442,40.299,157.533
C03239=1034.465,-27.962,-84.671,168.439,40.299,157.533
C03240=1034.459,-28.211,-84.658,168.437,40.300,157.533
C03241=1034.452,-28.461,-84.644,168.434,40.300,157.533
C03242=1034.446,-28.710,-84.631,168.433,40.301,157.533
C03243=1034.440,-28.959,-84.618,168.429,40.301,157.533
C03244=1034.433,-29.209,-84.604,168.428,40.302,157.533
C03245=1034.427,-29.459,-84.591,168.425,40.303,157.533
C03246=1034.420,-29.708,-84.578,168.423,40.303,157.533
C03247=1034.414,-29.957,-84.564,168.420,40.304,157.533
C03248=1034.407,-30.207,-84.551,168.418,40.305,157.533
C03249=1034.401,-30.457,-84.538,168.415,40.305,157.533
C03250=1034.395,-30.706,-84.525,168.413,40.305,157.533
C03251=1034.389,-30.957,-84.511,168.410,40.306,157.533
C03252=1034.383,-31.206,-84.497,168.408,40.306,157.533
C03253=1034.377,-31.455,-84.484,168.405,40.307,157.533
C03254=1034.371,-31.704,-84.471,168.403,40.307,157.533
C03255=1034.364,-31.955,-84.458,168.400,40.308,157.533
C03256=1034.358,-32.204,-84.445,168.398,40.308,157.533
C03257=1034.352,-32.453,-84.431,168.395,40.309,157.533
C03258=1034.345,-32.703,-84.418,168.392,40.310,157.533
C03259=1034.339,-32.953,-84.404,168.390,40.311,157.533
C03260=1034.333,-33.203,-84.392,168.387,40.311,157.533
C03261=1034.326,-33.452,-84.379,168.385,40.312,157.533
C03262=1034.320,-33.701,-84.365,168.382,40.312,157.533
C03263=1034.313,-33.951,-84.352,168.380,40.313,157.533
C03264=1034.308,-34.201,-84.339,168.377,40.313,157.533
C03265=1034.301,-34.450,-84.326,168.375,40.314,157.533
C03266=1034.295,-34.700,-84.313,168.372,40.314,157.533
C03267=1034.289,-34.949,-84.299,168.370,40.315,157.533
C03268=1034.282,-35.199,-84.286,168.367,40.315,157.533
C03269=1034.276,-35.449,-84.273,168.366,40.316,157.533
C03270=1034.269,-35.729,-84.259,168.363,40.317,157.533
C03271=1034.262,-36.010,-84.243,168.360,40.318,157.533
C03272=1034.255,-36.292,-84.229,168.357,40.318,157.533
C03273=1034.248,-36.572,-84.214,168.354,40.319,157.533
C03274=1034.242,-36.822,-84.202,168.352,40.319,157.533
C03275=1034.235,-37.072,-84.188,168.349,40.320,157.533
C03276=1034.229,-37.321,-84.175,168.347,40.320,157.533
C03277=1034.223,-37.571,-84.162,168.344,40.321,157.533
C03278=1034.217,-37.820,-84.149,168.342,40.321,157.533
C03279=1034.211,-38.070,-84.136,168.339,40.322,157.533
C03280=1034.205,-38.319,-84.123,168.337,40.322,157.533
C03281=1034.199,-38.569,-84.110,168.334,40.323,157.533
C03282=1034.193,-38.819,-84.097,168.332,40.324,157.533
C03283=1034.186,-39.068,-84.084,168.329,40.325,157.533
C03284=1034.180,-39.318,-84.071,168.326,40.325,157.533
C03285=1034.174,-39.568,-84.058,168.324,40.326,157.533
C03286=1034.167,-39.817,-84.046,168.321,40.327,157.533
C03287=1034.161,-40.066,-84.033,168.319,40.327,157.533
C03288=1034.155,-40.316,-84.020,168.316,40.328,157.533
C03289=1034.149,-40.566,-84.007,168.313,40.328,157.533
C03290=1034.142,-40.815,-83.995,168.311,40.329,157.533
C03291=1034.135,-41.065,-83.981,168.309,40.330,157.533
C03292=1034.129,-41.315,-83.969,168.307,40.330,157.533
C03293=1034.123,-41.564,-83.955,168.304,40.331,157.533
C03294=1034.117,-41.814,-83.943,168.301,40.332,157.533
C03295=1034.111,-42.064,-83.931,168.299,40.332,157.533
C03296=1034.104,-42.313,-83.918,168.296,40.333,157.533
C03297=1034.099,-42.563,-83.905,168.294,40.333,157.533
C03298=1034.092,-42.812,-83.892,168.291,40.334,157.533
C03299=1034.086,-43.062,-83.880,168.288,40.335,157.533
C03300=1034.079,-43.311,-83.866,168.286,40.336,157.533
C03301=1034.074,-43.561,-83.854,168.283,40.336,157.533
C03302=1034.067,-43.810,-83.842,168.281,40.337,157.533
C03303=1034.061,-44.060,-83.829,168.278,40.338,157.533
C03304=1034.055,-44.310,-83.816,168.275,40.339,157.533
C03305=1034.048,-44.560,-83.804,168.273,40.339,157.533
C03306=1034.041,-44.809,-83.791,168.270,40.340,157.533
C03307=1034.035,-45.059,-83.778,168.269,40.341,157.533
C03308=1034.030,-45.309,-83.765,168.265,40.341,157.533
C03309=1034.023,-45.558,-83.753,168.263,40.342,157.533
C03310=1034.017,-45.808,-83.740,168.261,40.343,157.533
C03311=1034.011,-46.058,-83.728,168.258,40.343,157.533
C03312=1034.004,-46.307,-83.715,168.256,40.344,157.533
C03313=1033.998,-46.556,-83.702,168.253,40.344,157.533
C03314=1033.992,-46.806,-83.690,168.250,40.345,157.533
C03315=1033.987,-47.056,-83.678,168.248,40.346,157.533
C03316=1033.980,-47.304,-83.665,168.245,40.346,157.533
C03317=1033.974,-47.554,-83.652,168.243,40.347,157.533
C03318=1033.968,-47.804,-83.640,168.240,40.348,157.533
C03319=1033.961,-48.054,-83.628,168.237,40.348,157.533
C03320=1033.955,-48.303,-83.615,168.235,40.349,157.533
C03321=1033.949,-48.553,-83.602,168.232,40.350,157.533
C03322=1033.942,-48.803,-83.590,168.229,40.351,157.533
C03323=1033.937,-49.052,-83.578,168.227,40.351,157.533
C03324=1033.931,-49.302,-83.565,168.224,40.352,157.533
C03325=1033.924,-49.552,-83.552,168.223,40.353,157.533
C03326=1033.918,-49.801,-83.540,168.220,40.354,157.533
C03327=1033.912,-50.051,-83.527,168.217,40.354,157.533
C03328=1033.906,-50.301,-83.515,168.215,40.355,157.533
C03329=1033.899,-50.550,-83.503,168.212,40.355,157.533
C03330=1033.894,-50.800,-83.491,168.209,40.356,157.533
C03331=1033.887,-51.049,-83.479,168.207,40.357,157.533
C03332=1033.881,-51.299,-83.467,168.204,40.358,157.533
C03333=1033.875,-51.548,-83.453,168.201,40.359,157.534
C03334=1033.867,-51.830,-83.440,168.198,40.360,157.534
C03335=1033.860,-52.112,-83.427,168.195,40.361,157.534
C03336=1033.853,-52.393,-83.412,168.192,40.362,157.534
C03337=1033.845,-52.674,-83.399,168.190,40.363,157.534
C03338=1033.839,-52.924,-83.387,168.188,40.363,157.534
C03339=1033.833,-53.174,-83.375,168.185,40.364,157.534
C03340=1033.826,-53.423,-83.363,168.182,40.365,157.534
C03341=1033.821,-53.672,-83.351,168.179,40.366,157.534
C03342=1033.814,-53.922,-83.339,168.177,40.367,157.534
C03343=1033.807,-54.172,-83.327,168.174,40.367,157.534
C03344=1033.801,-54.422,-83.314,168.171,40.368,157.534
C03345=1033.795,-54.671,-83.302,168.169,40.369,157.534
C03346=1033.788,-54.921,-83.290,168.166,40.370,157.534
C03347=1033.782,-55.171,-83.278,168.163,40.371,157.534
C03348=1033.776,-55.420,-83.266,168.160,40.372,157.534
C03349=1033.770,-55.670,-83.255,168.159,40.372,157.534
C03350=1033.764,-55.919,-83.242,168.156,40.373,157.534
C03351=1033.757,-56.169,-83.230,168.153,40.374,157.534
C03352=1033.751,-56.419,-83.218,168.151,40.375,157.534
C03353=1033.744,-56.668,-83.206,168.148,40.376,157.534
C03354=1033.738,-56.918,-83.194,168.145,40.377,157.534
C03355=1033.732,-57.167,-83.182,168.142,40.377,157.534
C03356=1033.725,-57.417,-83.170,168.140,40.378,157.534
C03357=1033.720,-57.667,-83.159,168.137,40.379,157.534
C03358=1033.713,-57.917,-83.147,168.134,40.380,157.534
C03359=1033.707,-58.166,-83.135,168.133,40.381,157.534
C03360=1033.700,-58.415,-83.123,168.130,40.382,157.534
C03361=1033.695,-58.665,-83.110,168.127,40.383,157.535
C03362=1033.688,-58.915,-83.099,168.124,40.384,157.535
C03363=1033.682,-59.165,-83.087,168.122,40.384,157.535
C03364=1033.676,-59.414,-83.075,168.119,40.385,157.535
C03365=1033.670,-59.663,-83.063,168.116,40.386,157.535
C03366=1033.663,-59.914,-83.052,168.114,40.387,157.535
C03367=1033.657,-60.163,-83.040,168.111,40.388,157.535
C03368=1033.651,-60.413,-83.027,168.108,40.389,157.535
C03369=1033.645,-60.662,-83.016,168.106,40.390,157.535
C03370=1033.638,-60.912,-83.005,168.103,40.390,157.535
C03371=1033.632,-61.162,-82.993,168.101,40.391,157.535
C03372=1033.626,-61.411,-82.980,168.098,40.392,157.535
C03373=1033.620,-61.660,-82.968,168.096,40.393,157.535
C03374=1033.613,-61.911,-82.957,168.093,40.394,157.535
C03375=1033.607,-62.161,-82.945,168.090,40.395,157.535
C03376=1033.601,-62.409,-82.933,168.087,40.396,157.535
C03377=1033.595,-62.660,-82.922,168.085,40.397,157.535
C03378=1033.588,-62.909,-82.910,168.082,40.397,157.535
C03379=1033.583,-63.158,-82.898,168.079,40.398,157.535
C03380=1033.577,-63.409,-82.886,168.076,40.399,157.535
C03381=1033.570,-63.658,-82.874,168.075,40.400,157.535
C03382=1033.564,-63.908,-82.864,168.072,40.401,157.535
C03383=1033.559,-64.158,-82.851,168.069,40.402,157.535
C03384=1033.552,-64.407,-82.839,168.066,40.403,157.535
C03385=1033.546,-64.657,-82.828,168.064,40.403,157.535
C03386=1033.539,-64.906,-82.816,168.061,40.404,157.535
C03387=1033.534,-65.157,-82.804,168.058,40.405,157.535
C03388=1033.528,-65.406,-82.793,168.056,40.406,157.535
C03389=1033.521,-65.655,-82.781,168.053,40.407,157.535
C03390=1033.515,-65.905,-82.770,168.050,40.407,157.535
C03391=1033.509,-66.154,-82.758,168.047,40.408,157.536
C03392=1033.503,-66.405,-82.746,168.046,40.409,157.536
C03393=1033.497,-66.654,-82.735,168.043,40.410,157.536
C03394=1033.491,-66.904,-82.723,168.040,40.411,157.536
C03395=1033.485,-67.153,-82.712,168.037,40.412,157.536
C03396=1033.479,-67.403,-82.700,168.035,40.412,157.536
C03397=1033.473,-67.653,-82.688,168.032,40.413,157.536
C03398=1033.466,-67.935,-82.675,168.029,40.414,157.536
C03399=1033.459,-68.218,-82.662,168.026,40.415,157.536
C03400=1033.452,-68.501,-82.649,168.023,40.416,157.536
C03401=1033.446,-68.783,-82.636,168.019,40.417,157.536
C03402=1033.439,-69.033,-82.624,168.018,40.418,157.536
C03403=1033.433,-69.282,-82.613,168.015,40.419,157.536
C03404=1033.427,-69.533,-82.602,168.012,40.420,157.536
C03405=1033.421,-69.781,-82.590,168.009,40.421,157.536
C03406=1033.415,-70.032,-82.578,168.007,40.422,157.536
C03407=1033.409,-70.281,-82.567,168.004,40.422,157.536
C03408=1033.403,-70.531,-82.556,168.001,40.423,157.536
C03409=1033.397,-70.781,-82.545,167.998,40.424,157.536
C03410=1033.390,-71.030,-82.533,167.996,40.425,157.536
C03411=1033.385,-71.280,-82.521,167.993,40.426,157.536
C03412=1033.379,-71.529,-82.509,167.990,40.427,157.536
C03413=1033.373,-71.779,-82.498,167.988,40.428,157.536
C03414=1033.367,-72.029,-82.487,167.986,40.429,157.536
C03415=1033.361,-72.278,-82.476,167.983,40.430,157.536
C03416=1033.355,-72.529,-82.464,167.980,40.430,157.536
C03417=1033.349,-72.778,-82.453,167.977,40.431,157.536
C03418=1033.343,-73.027,-82.441,167.975,40.432,157.536
C03419=1033.337,-73.277,-82.430,167.972,40.433,157.536
C03420=1033.331,-73.527,-82.419,167.969,40.434,157.536
C03421=1033.325,-73.777,-82.408,167.966,40.435,157.537
C03422=1033.320,-74.026,-82.396,167.964,40.436,157.537
C03423=1033.313,-74.276,-82.384,167.962,40.437,157.537
C03424=1033.307,-74.525,-82.374,167.959,40.438,157.537
C03425=1033.300,-74.776,-82.363,167.956,40.439,157.537
C03426=1033.294,-75.024,-82.351,167.953,40.440,157.537
C03427=1033.288,-75.275,-82.340,167.951,40.441,157.537
C03428=1033.282,-75.524,-82.329,167.948,40.441,157.537
C03429=1033.276,-75.774,-82.318,167.945,40.442,157.537
C03430=1033.270,-76.024,-82.307,167.942,40.443,157.537
C03431=1033.264,-76.273,-82.296,167.939,40.444,157.537
///RCONF 1,0,0,1,0,0,0,0,0,0,0,0,0,0,0,0,0,0,0,0,0,0,0,0
C03432=1033.258,-76.523,-82.285,167.937,40.446,157.537
C03433=1033.252,-76.772,-82.273,167.935,40.447,157.537
C03434=1033.246,-77.022,-82.262,167.932,40.448,157.537
C03435=1033.239,-77.272,-82.252,167.929,40.449,157.537
C03436=1033.233,-77.521,-82.241,167.926,40.450,157.537
C03437=1033.227,-77.771,-82.230,167.923,40.451,157.537
C03438=1033.221,-78.021,-82.219,167.920,40.452,157.537
C03439=1033.215,-78.271,-82.208,167.918,40.453,157.537
C03440=1033.209,-78.521,-82.197,167.916,40.454,157.537
C03441=1033.204,-78.770,-82.186,167.913,40.455,157.538
C03442=1033.197,-79.020,-82.175,167.910,40.456,157.538
C03443=1033.191,-79.270,-82.164,167.907,40.457,157.538
C03444=1033.185,-79.519,-82.153,167.905,40.458,157.538
///RCONF 1,0,0,0,0,0,0,0,0,0,0,0,0,0,0,0,0,0,0,0,0,0,0,0
C03445=1033.179,-79.769,-82.142,167.902,40.459,157.538
C03446=1033.173,-80.019,-82.131,167.899,40.460,157.538
C03447=1033.167,-80.269,-82.120,167.896,40.461,157.538
C03448=1033.160,-80.518,-82.110,167.894,40.462,157.538
C03449=1033.154,-80.767,-82.099,167.891,40.464,157.538
C03450=1033.148,-81.018,-82.088,167.888,40.465,157.538
C03451=1033.142,-81.267,-82.077,167.885,40.466,157.538
C03452=1033.136,-81.516,-82.067,167.883,40.467,157.538
C03453=1033.129,-81.766,-82.055,167.880,40.468,157.538
C03454=1033.123,-82.016,-82.045,167.877,40.469,157.538
C03455=1033.117,-82.265,-82.034,167.875,40.470,157.538
C03456=1033.110,-82.516,-82.024,167.872,40.472,157.539
C03457=1033.105,-82.765,-82.013,167.869,40.473,157.539
C03458=1033.099,-83.015,-82.002,167.866,40.474,157.539
C03459=1033.092,-83.264,-81.992,167.863,40.475,157.539
C03460=1033.086,-83.514,-81.981,167.861,40.476,157.539
C03461=1033.080,-83.763,-81.970,167.859,40.477,157.539
C03462=1033.073,-84.049,-81.958,167.855,40.479,157.539
C03463=1033.066,-84.333,-81.946,167.852,40.480,157.539
C03464=1033.059,-84.618,-81.934,167.849,40.481,157.539
C03465=1033.052,-84.903,-81.922,167.845,40.483,157.539
C03466=1033.046,-85.153,-81.911,167.843,40.483,157.539
C03467=1033.040,-85.402,-81.900,167.840,40.484,157.539
C03468=1033.034,-85.652,-81.891,167.838,40.486,157.540
C03469=1033.028,-85.902,-81.880,167.835,40.487,157.540
C03470=1033.021,-86.151,-81.869,167.832,40.488,157.540
C03471=1033.015,-86.401,-81.858,167.829,40.490,157.540
C03472=1033.010,-86.651,-81.848,167.826,40.491,157.540
C03473=1033.003,-86.901,-81.838,167.823,40.492,157.540
C03474=1032.997,-87.150,-81.827,167.821,40.493,157.540
C03475=1032.991,-87.400,-81.817,167.819,40.494,157.540
C03476=1032.985,-87.650,-81.806,167.816,40.495,157.540
C03477=1032.979,-87.900,-81.795,167.813,40.496,157.540
C03478=1032.973,-88.150,-81.786,167.810,40.498,157.540
C03479=1032.967,-88.399,-81.775,167.807,40.499,157.540
C03480=1032.961,-88.648,-81.764,167.804,40.500,157.540
C03481=1032.955,-88.898,-81.754,167.802,40.501,157.541
C03482=1032.949,-89.147,-81.744,167.799,40.502,157.541
C03483=1032.942,-89.398,-81.733,167.796,40.503,157.541
C03484=1032.937,-89.648,-81.723,167.793,40.505,157.541
C03485=1032.930,-89.897,-81.712,167.791,40.506,157.541
C03486=1032.925,-90.146,-81.701,167.788,40.507,157.541
C03487=1032.918,-90.396,-81.692,167.785,40.508,157.541
C03488=1032.913,-90.646,-81.681,167.783,40.509,157.541
C03489=1032.906,-90.896,-81.671,167.780,40.510,157.541
C03490=1032.900,-91.146,-81.660,167.777,40.511,157.541
C03491=1032.894,-91.395,-81.649,167.774,40.513,157.541
C03492=1032.888,-91.645,-81.640,167.771,40.514,157.541
C03493=1032.883,-91.895,-81.629,167.768,40.515,157.541
C03494=1032.876,-92.144,-81.619,167.766,40.517,157.542
C03495=1032.871,-92.394,-81.608,167.764,40.517,157.542
C03496=1032.864,-92.644,-81.599,167.761,40.518,157.542
C03497=1032.859,-92.893,-81.588,167.758,40.520,157.542
C03498=1032.853,-93.143,-81.578,167.755,40.521,157.542
C03499=1032.846,-93.393,-81.567,167.752,40.522,157.542
C03500=1032.840,-93.643,-81.558,167.750,40.524,157.542
C03501=1032.834,-93.892,-81.547,167.747,40.525,157.542
C03502=1032.829,-94.142,-81.536,167.744,40.526,157.542
C03503=1032.822,-94.392,-81.526,167.741,40.527,157.542
C03504=1032.817,-94.642,-81.516,167.738,40.528,157.542
C03505=1032.810,-94.891,-81.506,167.735,40.529,157.542
C03506=1032.805,-95.141,-81.496,167.733,40.530,157.542
C03507=1032.799,-95.391,-81.486,167.731,40.532,157.543
C03508=1032.793,-95.640,-81.475,167.728,40.533,157.543
C03509=1032.787,-95.890,-81.466,167.725,40.534,157.543
C03510=1032.781,-96.140,-81.455,167.722,40.535,157.543
C03511=1032.775,-96.389,-81.445,167.719,40.536,157.543
C03512=1032.770,-96.640,-81.435,167.716,40.537,157.543
C03513=1032.763,-96.889,-81.425,167.714,40.539,157.543
C03514=1032.758,-97.139,-81.415,167.711,40.540,157.543
C03515=1032.751,-97.388,-81.404,167.708,40.541,157.543
C03516=1032.746,-97.638,-81.394,167.705,40.543,157.543
C03517=1032.740,-97.888,-81.385,167.702,40.544,157.543
C03518=1032.733,-98.138,-81.375,167.699,40.545,157.543
C03519=1032.728,-98.387,-81.364,167.697,40.546,157.544
C03520=1032.722,-98.637,-81.355,167.695,40.548,157.544
C03521=1032.715,-98.887,-81.345,167.692,40.549,157.544
C03522=1032.710,-99.137,-81.335,167.689,40.550,157.544
C03523=1032.703,-99.386,-81.324,167.686,40.552,157.544
C03524=1032.697,-99.636,-81.315,167.683,40.553,157.544
C03525=1032.691,-99.886,-81.305,167.681,40.555,157.544
C03526=1032.685,-100.173,-81.294,167.677,40.556,157.544
C03527=1032.678,-100.460,-81.283,167.674,40.557,157.544
C03528=1032.671,-100.747,-81.271,167.670,40.559,157.545
C03529=1032.664,-101.034,-81.261,167.668,40.561,157.545
C03530=1032.658,-101.283,-81.250,167.665,40.562,157.545
C03531=1032.652,-101.533,-81.240,167.662,40.563,157.545
C03532=1032.646,-101.783,-81.231,167.659,40.564,157.545
C03533=1032.640,-102.033,-81.221,167.656,40.566,157.545
C03534=1032.634,-102.283,-81.211,167.653,40.567,157.545
C03535=1032.628,-102.533,-81.201,167.651,40.569,157.545
C03536=1032.622,-102.782,-81.192,167.648,40.570,157.545
C03537=1032.615,-103.032,-81.181,167.645,40.571,157.545
C03538=1032.609,-103.281,-81.172,167.642,40.572,157.545
C03539=1032.604,-103.531,-81.162,167.639,40.574,157.546
C03540=1032.598,-103.781,-81.152,167.637,40.576,157.546
C03541=1032.592,-104.030,-81.143,167.634,40.577,157.546
C03542=1032.586,-104.280,-81.133,167.631,40.578,157.546
C03543=1032.580,-104.530,-81.123,167.628,40.579,157.546
C03544=1032.574,-104.780,-81.114,167.625,40.581,157.546
C03545=1032.568,-105.030,-81.104,167.622,40.582,157.546
C03546=1032.562,-105.280,-81.094,167.621,40.584,157.546
C03547=1032.556,-105.529,-81.085,167.618,40.585,157.547
C03548=1032.551,-105.779,-81.075,167.615,40.586,157.547
C03549=1032.545,-106.029,-81.066,167.612,40.588,157.547
C03550=1032.538,-106.279,-81.056,167.609,40.589,157.547
C03551=1032.532,-106.528,-81.046,167.607,40.590,157.547
C03552=1032.526,-106.778,-81.037,167.604,40.592,157.547
C03553=1032.521,-107.027,-81.028,167.601,40.593,157.547
C03554=1032.514,-107.277,-81.018,167.598,40.595,157.547
C03555=1032.509,-107.527,-81.008,167.595,40.596,157.547
C03556=1032.503,-107.777,-80.998,167.593,40.597,157.547
C03557=1032.497,-108.027,-80.989,167.590,40.599,157.548
C03558=1032.491,-108.276,-80.980,167.587,40.600,157.548
C03559=1032.485,-108.526,-80.971,167.584,40.602,157.548
C03560=1032.479,-108.776,-80.961,167.581,40.603,157.548
C03561=1032.473,-109.026,-80.952,167.579,40.605,157.548
C03562=1032.467,-109.276,-80.942,167.576,40.606,157.548
C03563=1032.461,-109.525,-80.933,167.573,40.608,157.548
C03564=1032.455,-109.775,-80.923,167.570,40.609,157.548
C03565=1032.449,-110.024,-80.914,167.566,40.610,157.548
C03566=1032.443,-110.275,-80.905,167.564,40.612,157.549
C03567=1032.437,-110.524,-80.896,167.561,40.614,157.549
C03568=1032.431,-110.774,-80.886,167.558,40.615,157.549
C03569=1032.425,-111.023,-80.877,167.555,40.616,157.549
C03570=1032.419,-111.273,-80.867,167.553,40.618,157.549
C03571=1032.414,-111.523,-80.858,167.550,40.620,157.549
C03572=1032.407,-111.773,-80.849,167.547,40.621,157.549
C03573=1032.401,-112.023,-80.839,167.544,40.622,157.549
C03574=1032.395,-112.272,-80.830,167.541,40.624,157.550
C03575=1032.390,-112.522,-80.821,167.539,40.626,157.550
C03576=1032.384,-112.772,-80.812,167.536,40.627,157.550
C03577=1032.377,-113.022,-80.802,167.533,40.628,157.550
C03578=1032.372,-113.271,-80.794,167.530,40.630,157.550
C03579=1032.366,-113.521,-80.784,167.527,40.631,157.550
C03580=1032.360,-113.771,-80.775,167.525,40.633,157.550
C03581=1032.354,-114.020,-80.765,167.522,40.634,157.550
C03582=1032.348,-114.270,-80.756,167.519,40.636,157.551
C03583=1032.342,-114.520,-80.747,167.516,40.637,157.551
C03584=1032.337,-114.769,-80.738,167.513,40.639,157.551
C03585=1032.331,-115.020,-80.729,167.511,40.640,157.551
C03586=1032.325,-115.270,-80.719,167.508,40.642,157.551
C03587=1032.319,-115.519,-80.711,167.505,40.644,157.551
C03588=1032.312,-115.769,-80.702,167.503,40.645,157.551
C03589=1032.306,-116.019,-80.692,167.500,40.646,157.551
C03590=1032.300,-116.305,-80.682,167.496,40.648,157.552
C03591=1032.293,-116.591,-80.672,167.493,40.650,157.552
C03592=1032.286,-116.878,-80.661,167.489,40.652,157.552
C03593=1032.280,-117.165,-80.650,167.487,40.654,157.552
